   1:L PR[91] R[100]mm/sec CNT100;
   1:  PR[91,1] = PR[90,1] + 32.594;
   1:  PR[91,2] = PR[90,2] + 13.699;
   1:L PR[91] R[100]mm/sec CNT100;
   1:  PR[91,1] = PR[90,1] + 30.652;
   1:  PR[91,2] = PR[90,2] + 14.958;
   1:L PR[91] R[100]mm/sec CNT100;
   1:  PR[91,1] = PR[90,1] + 29.155;
   1:  PR[91,2] = PR[90,2] + 15.871;
   1:L PR[91] R[100]mm/sec CNT100;
   1:  PR[91,1] = PR[90,1] + 26.400;
   1:  PR[91,2] = PR[90,2] + 16.913;
   1:L PR[91] R[100]mm/sec CNT100;
   1:  PR[91,1] = PR[90,1] + 25.342;
   1:  PR[91,2] = PR[90,2] + 17.273;
   1:L PR[91] R[100]mm/sec CNT100;
   1:  PR[91,1] = PR[90,1] + 21.693;
   1:  PR[91,2] = PR[90,2] + 17.818;
   1:L PR[91] R[100]mm/sec CNT100;
   1:  PR[91,1] = PR[90,1] + 21.351;
   1:  PR[91,2] = PR[90,2] + 17.856;
   1:L PR[91] R[100]mm/sec CNT100;
   1:  PR[91,1] = PR[90,1] + 18.415;
   1:  PR[91,2] = PR[90,2] + 17.666;
   1:L PR[91] R[100]mm/sec CNT100;
   1:  PR[91,1] = PR[90,1] + 17.180;
   1:  PR[91,2] = PR[90,2] + 17.601;
   1:L PR[91] R[100]mm/sec CNT100;
   1:  PR[91,1] = PR[90,1] + 13.479;
   1:  PR[91,2] = PR[90,2] + 16.611;
   1:L PR[91] R[100]mm/sec CNT100;
   1:  PR[91,1] = PR[90,1] + 13.072;
   1:  PR[91,2] = PR[90,2] + 16.479;
   1:L PR[91] R[100]mm/sec CNT100;
   1:  PR[91,1] = PR[90,1] + 10.503;
   1:  PR[91,2] = PR[90,2] + 15.153;
   1:L PR[91] R[100]mm/sec CNT100;
   1:  PR[91,1] = PR[90,1] + 9.678;
   1:  PR[91,2] = PR[90,2] + 14.763;
   1:L PR[91] R[100]mm/sec CNT100;
   1:  PR[91,1] = PR[90,1] + 8.783;
   1:  PR[91,2] = PR[90,2] + 14.163;
   1:L PR[91] R[100]mm/sec CNT100;
   1:  PR[91,1] = PR[90,1] + 7.210;
   1:  PR[91,2] = PR[90,2] + 12.860;
   1:L PR[91] R[100]mm/sec CNT100;
   1:  PR[91,1] = PR[90,1] + 6.133;
   1:  PR[91,2] = PR[90,2] + 11.895;
   1:L PR[91] R[100]mm/sec CNT100;
   1:  PR[91,1] = PR[90,1] + 4.893;
   1:  PR[91,2] = PR[90,2] + 10.402;
   1:L PR[91] R[100]mm/sec CNT100;
   1:  PR[91,1] = PR[90,1] + 4.050;
   1:  PR[91,2] = PR[90,2] + 9.302;
   1:L PR[91] R[100]mm/sec CNT100;
   1:  PR[91,1] = PR[90,1] + 3.471;
   1:  PR[91,2] = PR[90,2] + 8.699;
   1:L PR[91] R[100]mm/sec CNT100;
   1:  PR[91,1] = PR[90,1] + 2.632;
   1:  PR[91,2] = PR[90,2] + 8.134;
   1:L PR[91] R[100]mm/sec CNT100;
   1:  PR[91,1] = PR[90,1] + 1.785;
   1:  PR[91,2] = PR[90,2] + 7.929;
   1:L PR[91] R[100]mm/sec CNT100;
   1:  PR[91,1] = PR[90,1] + 1.392;
   1:  PR[91,2] = PR[90,2] + 7.757;
   1:L PR[91] R[100]mm/sec CNT100;
   1:  PR[91] = PR[90];
   1:  PR[91,1] = PR[90,1] + -1.445;
   1:  PR[91,2] = PR[90,2] + 8.302;
   1:  PR[91,3] = PR[90,3] + 22.295;
   1:L PR[91] R[100]mm/sec CNT100;
   1:  PR[91,1] = PR[90,1] + -2.877;
   1:  PR[91,2] = PR[90,2] + 8.645;
   1:L PR[91] R[100]mm/sec CNT100;
   1:  PR[91,1] = PR[90,1] + -3.773;
   1:  PR[91,2] = PR[90,2] + 9.251;
   1:L PR[91] R[100]mm/sec CNT100;
   1:  PR[91,1] = PR[90,1] + -4.266;
   1:  PR[91,2] = PR[90,2] + 9.782;
   1:L PR[91] R[100]mm/sec CNT100;
   1:  PR[91,1] = PR[90,1] + -6.077;
   1:  PR[91,2] = PR[90,2] + 11.940;
   1:L PR[91] R[100]mm/sec CNT100;
   1:  PR[91,1] = PR[90,1] + -8.345;
   1:  PR[91,2] = PR[90,2] + 13.932;
   1:L PR[91] R[100]mm/sec CNT100;
   1:  PR[91,1] = PR[90,1] + -10.027;
   1:  PR[91,2] = PR[90,2] + 15.061;
   1:L PR[91] R[100]mm/sec CNT100;
   1:  PR[91,1] = PR[90,1] + -11.357;
   1:  PR[91,2] = PR[90,2] + 15.744;
   1:L PR[91] R[100]mm/sec CNT100;
   1:  PR[91,1] = PR[90,1] + -12.975;
   1:  PR[91,2] = PR[90,2] + 16.525;
   1:L PR[91] R[100]mm/sec CNT100;
   1:  PR[91,1] = PR[90,1] + -14.146;
   1:  PR[91,2] = PR[90,2] + 16.905;
   1:L PR[91] R[100]mm/sec CNT100;
   1:  PR[91,1] = PR[90,1] + -16.672;
   1:  PR[91,2] = PR[90,2] + 17.580;
   1:L PR[91] R[100]mm/sec CNT100;
   1:  PR[91,1] = PR[90,1] + -17.455;
   1:  PR[91,2] = PR[90,2] + 17.722;
   1:L PR[91] R[100]mm/sec CNT100;
   1:  PR[91,1] = PR[90,1] + -21.155;
   1:  PR[91,2] = PR[90,2] + 17.918;
   1:L PR[91] R[100]mm/sec CNT100;
   1:  PR[91,1] = PR[90,1] + -21.482;
   1:  PR[91,2] = PR[90,2] + 17.931;
   1:L PR[91] R[100]mm/sec CNT100;
   1:  PR[91,1] = PR[90,1] + -21.616;
   1:  PR[91,2] = PR[90,2] + 17.919;
   1:L PR[91] R[100]mm/sec CNT100;
   1:  PR[91,1] = PR[90,1] + -25.669;
   1:  PR[91,2] = PR[90,2] + 17.290;
   1:L PR[91] R[100]mm/sec CNT100;
   1:  PR[91,1] = PR[90,1] + -29.492;
   1:  PR[91,2] = PR[90,2] + 15.850;
   1:L PR[91] R[100]mm/sec CNT100;
   1:  PR[91,1] = PR[90,1] + -30.051;
   1:  PR[91,2] = PR[90,2] + 15.509;
   1:L PR[91] R[100]mm/sec CNT100;
   1:  PR[91,1] = PR[90,1] + -32.898;
   1:  PR[91,2] = PR[90,2] + 13.662;
   1:L PR[91] R[100]mm/sec CNT100;
   1:  PR[91,1] = PR[90,1] + -33.763;
   1:  PR[91,2] = PR[90,2] + 12.821;
   1:L PR[91] R[100]mm/sec CNT100;
   1:  PR[91,1] = PR[90,1] + -35.755;
   1:  PR[91,2] = PR[90,2] + 10.797;
   1:L PR[91] R[100]mm/sec CNT100;
   1:  PR[91,1] = PR[90,1] + -36.625;
   1:  PR[91,2] = PR[90,2] + 9.444;
   1:L PR[91] R[100]mm/sec CNT100;
   1:  PR[91,1] = PR[90,1] + -37.914;
   1:  PR[91,2] = PR[90,2] + 7.364;
   1:L PR[91] R[100]mm/sec CNT100;
   1:  PR[91,1] = PR[90,1] + -39.261;
   1:  PR[91,2] = PR[90,2] + 3.606;
   1:L PR[91] R[100]mm/sec CNT100;
   1:  PR[91,1] = PR[90,1] + -39.495;
   1:  PR[91,2] = PR[90,2] + 1.583;
   1:L PR[91] R[100]mm/sec CNT100;
   1:  PR[91,1] = PR[90,1] + -39.753;
   1:  PR[91,2] = PR[90,2] + -0.438;
   1:L PR[91] R[100]mm/sec CNT100;
   1:  PR[91,1] = PR[90,1] + -39.620;
   1:  PR[91,2] = PR[90,2] + -1.583;
   1:L PR[91] R[100]mm/sec CNT100;
   1:  PR[91,1] = PR[90,1] + -39.489;
   1:  PR[91,2] = PR[90,2] + -2.382;
   1:L PR[91] R[100]mm/sec CNT100;
   1:  PR[91,1] = PR[90,1] + -39.258;
   1:  PR[91,2] = PR[90,2] + -4.463;
   1:L PR[91] R[100]mm/sec CNT100;
   1:  PR[91,1] = PR[90,1] + -38.549;
   1:  PR[91,2] = PR[90,2] + -6.462;
   1:L PR[91] R[100]mm/sec CNT100;
   1:  PR[91,1] = PR[90,1] + -37.916;
   1:  PR[91,2] = PR[90,2] + -8.208;
   1:L PR[91] R[100]mm/sec CNT100;
   1:  PR[91,1] = PR[90,1] + -36.624;
   1:  PR[91,2] = PR[90,2] + -10.292;
   1:L PR[91] R[100]mm/sec CNT100;
   1:  PR[91,1] = PR[90,1] + -35.754;
   1:  PR[91,2] = PR[90,2] + -11.645;
   1:L PR[91] R[100]mm/sec CNT100;
   1:  PR[91,1] = PR[90,1] + -33.761;
   1:  PR[91,2] = PR[90,2] + -13.670;
   1:L PR[91] R[100]mm/sec CNT100;
   1:  PR[91,1] = PR[90,1] + -32.896;
   1:  PR[91,2] = PR[90,2] + -14.510;
   1:L PR[91] R[100]mm/sec CNT100;
   1:  PR[91,1] = PR[90,1] + -30.048;
   1:  PR[91,2] = PR[90,2] + -16.357;
   1:L PR[91] R[100]mm/sec CNT100;
   1:  PR[91,1] = PR[90,1] + -29.490;
   1:  PR[91,2] = PR[90,2] + -16.698;
   1:L PR[91] R[100]mm/sec CNT100;
   1:  PR[91,1] = PR[90,1] + -25.665;
   1:  PR[91,2] = PR[90,2] + -18.138;
   1:L PR[91] R[100]mm/sec CNT100;
   1:  PR[91,1] = PR[90,1] + -21.611;
   1:  PR[91,2] = PR[90,2] + -18.766;
   1:L PR[91] R[100]mm/sec CNT100;
   1:  PR[91,1] = PR[90,1] + -21.494;
   1:  PR[91,2] = PR[90,2] + -18.777;
   1:L PR[91] R[100]mm/sec CNT100;
   1:  PR[91,1] = PR[90,1] + -18.062;
   1:  PR[91,2] = PR[90,2] + -18.588;
   1:L PR[91] R[100]mm/sec CNT100;
   1:  PR[91,1] = PR[90,1] + -17.432;
   1:  PR[91,2] = PR[90,2] + -18.565;
   1:L PR[91] R[100]mm/sec CNT100;
   1:  PR[91,1] = PR[90,1] + -16.667;
   1:  PR[91,2] = PR[90,2] + -18.427;
   1:L PR[91] R[100]mm/sec CNT100;
   1:  PR[91,1] = PR[90,1] + -14.143;
   1:  PR[91,2] = PR[90,2] + -17.751;
   1:L PR[91] R[100]mm/sec CNT100;
   1:  PR[91,1] = PR[90,1] + -13.004;
   1:  PR[91,2] = PR[90,2] + -17.381;
   1:L PR[91] R[100]mm/sec CNT100;
   1:  PR[91,1] = PR[90,1] + -11.460;
   1:  PR[91,2] = PR[90,2] + -16.582;
   1:L PR[91] R[100]mm/sec CNT100;
   1:  PR[91,1] = PR[90,1] + -9.994;
   1:  PR[91,2] = PR[90,2] + -15.886;
   1:L PR[91] R[100]mm/sec CNT100;
   1:  PR[91,1] = PR[90,1] + -8.315;
   1:  PR[91,2] = PR[90,2] + -14.758;
   1:L PR[91] R[100]mm/sec CNT100;
   1:  PR[91,1] = PR[90,1] + -7.791;
   1:  PR[91,2] = PR[90,2] + -14.325;
   1:L PR[91] R[100]mm/sec CNT100;
   1:  PR[91,1] = PR[90,1] + -6.085;
   1:  PR[91,2] = PR[90,2] + -12.797;
   1:L PR[91] R[100]mm/sec CNT100;
   1:  PR[91,1] = PR[90,1] + -4.272;
   1:  PR[91,2] = PR[90,2] + -10.633;
   1:L PR[91] R[100]mm/sec CNT100;
   1:  PR[91,1] = PR[90,1] + -3.791;
   1:  PR[91,2] = PR[90,2] + -10.110;
   1:L PR[91] R[100]mm/sec CNT100;
   1:  PR[91,1] = PR[90,1] + -2.878;
   1:  PR[91,2] = PR[90,2] + -9.493;
   1:L PR[91] R[100]mm/sec CNT100;
   1:  PR[91,1] = PR[90,1] + -1.445;
   1:  PR[91,2] = PR[90,2] + -9.149;
   1:L PR[91] R[100]mm/sec CNT100;
   1:  PR[91,1] = PR[90,1] + 0.974;
   1:L PR[91] R[100]mm/sec CNT100;
   1:  PR[91,1] = PR[90,1] + 2.406;
   1:  PR[91,2] = PR[90,2] + -9.492;
   1:L PR[91] R[100]mm/sec CNT100;
   1:  PR[91,1] = PR[90,1] + 3.303;
   1:  PR[91,2] = PR[90,2] + -10.098;
   1:L PR[91] R[100]mm/sec CNT100;
   1:  PR[91,1] = PR[90,1] + 3.795;
   1:  PR[91,2] = PR[90,2] + -10.630;
   1:L PR[91] R[100]mm/sec CNT100;
   1:  PR[91,1] = PR[90,1] + 5.623;
   1:  PR[91,2] = PR[90,2] + -12.812;
   1:L PR[91] R[100]mm/sec CNT100;
   1:  PR[91,1] = PR[90,1] + 7.885;
   1:  PR[91,2] = PR[90,2] + -14.797;
   1:L PR[91] R[100]mm/sec CNT100;
   1:  PR[91,1] = PR[90,1] + 9.546;
   1:  PR[91,2] = PR[90,2] + -15.911;
   1:L PR[91] R[100]mm/sec CNT100;
   1:  PR[91,1] = PR[90,1] + 10.876;
   1:  PR[91,2] = PR[90,2] + -16.592;
   1:L PR[91] R[100]mm/sec CNT100;
   1:  PR[91,1] = PR[90,1] + 12.490;
   1:  PR[91,2] = PR[90,2] + -17.369;
   1:L PR[91] R[100]mm/sec CNT100;
   1:  PR[91,1] = PR[90,1] + 13.666;
   1:  PR[91,2] = PR[90,2] + -17.751;
   1:L PR[91] R[100]mm/sec CNT100;
   1:  PR[91,1] = PR[90,1] + 16.194;
   1:  PR[91,2] = PR[90,2] + -18.427;
   1:L PR[91] R[100]mm/sec CNT100;
   1:  PR[91,1] = PR[90,1] + 16.977;
   1:  PR[91,2] = PR[90,2] + -18.570;
   1:L PR[91] R[100]mm/sec CNT100;
   1:  PR[91,1] = PR[90,1] + 21.019;
   1:  PR[91,2] = PR[90,2] + -18.777;
   1:L PR[91] R[100]mm/sec CNT100;
   1:  PR[91,1] = PR[90,1] + 21.138;
   1:  PR[91,2] = PR[90,2] + -18.767;
   1:L PR[91] R[100]mm/sec CNT100;
   1:  PR[91,1] = PR[90,1] + 25.192;
   1:  PR[91,2] = PR[90,2] + -18.135;
   1:L PR[91] R[100]mm/sec CNT100;
   1:  PR[91,1] = PR[90,1] + 29.016;
   1:  PR[91,2] = PR[90,2] + -16.696;
   1:L PR[91] R[100]mm/sec CNT100;
   1:  PR[91,1] = PR[90,1] + 29.575;
   1:  PR[91,2] = PR[90,2] + -16.355;
   1:L PR[91] R[100]mm/sec CNT100;
   1:  PR[91,1] = PR[90,1] + 32.419;
   1:  PR[91,2] = PR[90,2] + -14.511;
   1:L PR[91] R[100]mm/sec CNT100;
   1:  PR[91,1] = PR[90,1] + 33.282;
   1:  PR[91,2] = PR[90,2] + -13.671;
   1:L PR[91] R[100]mm/sec CNT100;
   1:  PR[91,1] = PR[90,1] + 35.275;
   1:  PR[91,2] = PR[90,2] + -11.638;
   1:L PR[91] R[100]mm/sec CNT100;
   1:  PR[91,1] = PR[90,1] + 36.146;
   1:  PR[91,2] = PR[90,2] + -10.284;
   1:L PR[91] R[100]mm/sec CNT100;
   1:  PR[91,1] = PR[90,1] + 37.435;
   1:  PR[91,2] = PR[90,2] + -8.207;
   1:L PR[91] R[100]mm/sec CNT100;
   1:  PR[91,1] = PR[90,1] + 38.781;
   1:  PR[91,2] = PR[90,2] + -4.466;
   1:L PR[91] R[100]mm/sec CNT100;
   1:  PR[91,1] = PR[90,1] + 39.015;
   1:  PR[91,2] = PR[90,2] + -2.439;
   1:L PR[91] R[100]mm/sec CNT100;
   1:  PR[91,1] = PR[90,1] + 39.273;
   1:  PR[91,2] = PR[90,2] + -0.410;
   1:L PR[91] R[100]mm/sec CNT100;
   1:  PR[91,1] = PR[90,1] + 39.140;
   1:  PR[91,2] = PR[90,2] + 0.741;
   1:L PR[91] R[100]mm/sec CNT100;
   1:  PR[91,1] = PR[90,1] + 39.009;
   1:  PR[91,2] = PR[90,2] + 1.541;
   1:L PR[91] R[100]mm/sec CNT100;
   1:  PR[91,1] = PR[90,1] + 38.779;
   1:  PR[91,2] = PR[90,2] + 3.625;
   1:L PR[91] R[100]mm/sec CNT100;
   1:  PR[91,1] = PR[90,1] + 37.435;
   1:  PR[91,2] = PR[90,2] + 7.361;
   1:L PR[91] R[100]mm/sec CNT100;
   1:  PR[91,1] = PR[90,1] + 36.146;
   1:  PR[91,2] = PR[90,2] + 9.437;
   1:L PR[91] R[100]mm/sec CNT100;
   1:  PR[91,1] = PR[90,1] + 35.274;
   1:  PR[91,2] = PR[90,2] + 10.792;
   1:L PR[91] R[100]mm/sec CNT100;
   1:  PR[91,1] = PR[90,1] + 33.281;
   1:  PR[91,2] = PR[90,2] + 12.823;
   1:L PR[91] R[100]mm/sec CNT100;
   1:  PR[91,1] = PR[90,1] + 32.418;
   1:  PR[91,2] = PR[90,2] + 13.665;
   1:L PR[91] R[100]mm/sec CNT100;
   1:  PR[91,1] = PR[90,1] + 29.574;
   1:  PR[91,2] = PR[90,2] + 15.508;
   1:L PR[91] R[100]mm/sec CNT100;
   1:  PR[91,1] = PR[90,1] + 29.015;
   1:  PR[91,2] = PR[90,2] + 15.849;
   1:L PR[91] R[100]mm/sec CNT100;
   1:  PR[91,1] = PR[90,1] + 25.191;
   1:  PR[91,2] = PR[90,2] + 17.288;
   1:L PR[91] R[100]mm/sec CNT100;
   1:  PR[91,1] = PR[90,1] + 21.137;
   1:  PR[91,2] = PR[90,2] + 17.919;
   1:L PR[91] R[100]mm/sec CNT100;
   1:  PR[91,1] = PR[90,1] + 21.021;
   1:  PR[91,2] = PR[90,2] + 17.930;
   1:L PR[91] R[100]mm/sec CNT100;
   1:  PR[91,1] = PR[90,1] + 17.586;
   1:  PR[91,2] = PR[90,2] + 17.742;
   1:L PR[91] R[100]mm/sec CNT100;
   1:  PR[91,1] = PR[90,1] + 16.959;
   1:  PR[91,2] = PR[90,2] + 17.719;
   1:L PR[91] R[100]mm/sec CNT100;
   1:  PR[91,1] = PR[90,1] + 16.193;
   1:  PR[91,2] = PR[90,2] + 17.580;
   1:L PR[91] R[100]mm/sec CNT100;
   1:  PR[91,1] = PR[90,1] + 13.666;
   1:  PR[91,2] = PR[90,2] + 16.903;
   1:L PR[91] R[100]mm/sec CNT100;
   1:  PR[91,1] = PR[90,1] + 12.521;
   1:  PR[91,2] = PR[90,2] + 16.532;
   1:L PR[91] R[100]mm/sec CNT100;
   1:  PR[91,1] = PR[90,1] + 10.976;
   1:  PR[91,2] = PR[90,2] + 15.735;
   1:L PR[91] R[100]mm/sec CNT100;
   1:  PR[91,1] = PR[90,1] + 9.515;
   1:  PR[91,2] = PR[90,2] + 15.043;
   1:L PR[91] R[100]mm/sec CNT100;
   1:  PR[91,1] = PR[90,1] + 7.856;
   1:  PR[91,2] = PR[90,2] + 13.930;
   1:L PR[91] R[100]mm/sec CNT100;
   1:  PR[91,1] = PR[90,1] + 7.329;
   1:  PR[91,2] = PR[90,2] + 13.494;
   1:L PR[91] R[100]mm/sec CNT100;
   1:  PR[91,1] = PR[90,1] + 5.632;
   1:  PR[91,2] = PR[90,2] + 11.974;
   1:L PR[91] R[100]mm/sec CNT100;
   1:  PR[91,1] = PR[90,1] + 3.802;
   1:  PR[91,2] = PR[90,2] + 9.786;
   1:L PR[91] R[100]mm/sec CNT100;
   1:  PR[91,1] = PR[90,1] + 3.320;
   1:  PR[91,2] = PR[90,2] + 9.263;
   1:L PR[91] R[100]mm/sec CNT100;
   1:  PR[91,1] = PR[90,1] + 2.407;
   1:  PR[91,2] = PR[90,2] + 8.645;
   1:L PR[91] R[100]mm/sec CNT100;
   1:  PR[91,1] = PR[90,1] + 0.974;
   1:  PR[91,2] = PR[90,2] + 8.302;
   1:L PR[91] R[100]mm/sec CNT100;
   1:  PR[91] = PR[90];
   1:  PR[91,1] = PR[90,1] + -1.220;
   1:  PR[91,2] = PR[90,2] + 8.847;
   1:  PR[91,3] = PR[90,3] + 23.595;
   1:L PR[91] R[100]mm/sec CNT100;
   1:  PR[91,1] = PR[90,1] + -2.655;
   1:  PR[91,2] = PR[90,2] + 9.172;
   1:L PR[91] R[100]mm/sec CNT100;
   1:  PR[91,1] = PR[90,1] + -3.468;
   1:  PR[91,2] = PR[90,2] + 9.721;
   1:L PR[91] R[100]mm/sec CNT100;
   1:  PR[91,1] = PR[90,1] + -3.995;
   1:  PR[91,2] = PR[90,2] + 10.252;
   1:L PR[91] R[100]mm/sec CNT100;
   1:  PR[91,1] = PR[90,1] + -5.523;
   1:  PR[91,2] = PR[90,2] + 12.037;
   1:L PR[91] R[100]mm/sec CNT100;
   1:  PR[91,1] = PR[90,1] + -5.576;
   1:  PR[91,2] = PR[90,2] + 12.090;
   1:L PR[91] R[100]mm/sec CNT100;
   1:  PR[91,1] = PR[90,1] + -7.560;
   1:  PR[91,2] = PR[90,2] + 13.830;
   1:L PR[91] R[100]mm/sec CNT100;
   1:  PR[91,1] = PR[90,1] + -9.831;
   1:  PR[91,2] = PR[90,2] + 15.322;
   1:L PR[91] R[100]mm/sec CNT100;
   1:  PR[91,1] = PR[90,1] + -12.430;
   1:  PR[91,2] = PR[90,2] + 16.580;
   1:L PR[91] R[100]mm/sec CNT100;
   1:  PR[91,1] = PR[90,1] + -14.335;
   1:  PR[91,2] = PR[90,2] + 17.199;
   1:L PR[91] R[100]mm/sec CNT100;
   1:  PR[91,1] = PR[90,1] + -15.650;
   1:  PR[91,2] = PR[90,2] + 17.550;
   1:L PR[91] R[100]mm/sec CNT100;
   1:  PR[91,1] = PR[90,1] + -17.281;
   1:  PR[91,2] = PR[90,2] + 17.845;
   1:L PR[91] R[100]mm/sec CNT100;
   1:  PR[91,1] = PR[90,1] + -19.601;
   1:  PR[91,2] = PR[90,2] + 17.968;
   1:L PR[91] R[100]mm/sec CNT100;
   1:  PR[91,1] = PR[90,1] + -20.896;
   1:  PR[91,2] = PR[90,2] + 18.020;
   1:L PR[91] R[100]mm/sec CNT100;
   1:  PR[91,1] = PR[90,1] + -21.739;
   1:  PR[91,2] = PR[90,2] + 17.943;
   1:L PR[91] R[100]mm/sec CNT100;
   1:  PR[91,1] = PR[90,1] + -24.981;
   1:  PR[91,2] = PR[90,2] + 17.433;
   1:L PR[91] R[100]mm/sec CNT100;
   1:  PR[91,1] = PR[90,1] + -25.369;
   1:  PR[91,2] = PR[90,2] + 17.344;
   1:L PR[91] R[100]mm/sec CNT100;
   1:  PR[91,1] = PR[90,1] + -29.281;
   1:  PR[91,2] = PR[90,2] + 15.858;
   1:L PR[91] R[100]mm/sec CNT100;
   1:  PR[91,1] = PR[90,1] + -32.702;
   1:  PR[91,2] = PR[90,2] + 13.640;
   1:L PR[91] R[100]mm/sec CNT100;
   1:  PR[91,1] = PR[90,1] + -35.550;
   1:  PR[91,2] = PR[90,2] + 10.758;
   1:L PR[91] R[100]mm/sec CNT100;
   1:  PR[91,1] = PR[90,1] + -35.885;
   1:  PR[91,2] = PR[90,2] + 10.237;
   1:L PR[91] R[100]mm/sec CNT100;
   1:  PR[91,1] = PR[90,1] + -37.684;
   1:  PR[91,2] = PR[90,2] + 7.334;
   1:L PR[91] R[100]mm/sec CNT100;
   1:  PR[91,1] = PR[90,1] + -39.018;
   1:  PR[91,2] = PR[90,2] + 3.596;
   1:L PR[91] R[100]mm/sec CNT100;
   1:  PR[91,1] = PR[90,1] + -39.146;
   1:  PR[91,2] = PR[90,2] + 2.487;
   1:L PR[91] R[100]mm/sec CNT100;
   1:  PR[91,1] = PR[90,1] + -39.518;
   1:  PR[91,2] = PR[90,2] + -0.432;
   1:L PR[91] R[100]mm/sec CNT100;
   1:  PR[91,1] = PR[90,1] + -39.342;
   1:  PR[91,2] = PR[90,2] + -1.502;
   1:L PR[91] R[100]mm/sec CNT100;
   1:  PR[91,1] = PR[90,1] + -39.015;
   1:  PR[91,2] = PR[90,2] + -4.451;
   1:L PR[91] R[100]mm/sec CNT100;
   1:  PR[91,1] = PR[90,1] + -38.002;
   1:  PR[91,2] = PR[90,2] + -7.308;
   1:L PR[91] R[100]mm/sec CNT100;
   1:  PR[91,1] = PR[90,1] + -37.687;
   1:  PR[91,2] = PR[90,2] + -8.176;
   1:L PR[91] R[100]mm/sec CNT100;
   1:  PR[91,1] = PR[90,1] + -35.884;
   1:  PR[91,2] = PR[90,2] + -11.086;
   1:L PR[91] R[100]mm/sec CNT100;
   1:  PR[91,1] = PR[90,1] + -35.549;
   1:  PR[91,2] = PR[90,2] + -11.607;
   1:L PR[91] R[100]mm/sec CNT100;
   1:  PR[91,1] = PR[90,1] + -32.701;
   1:  PR[91,2] = PR[90,2] + -14.487;
   1:L PR[91] R[100]mm/sec CNT100;
   1:  PR[91,1] = PR[90,1] + -29.241;
   1:  PR[91,2] = PR[90,2] + -16.720;
   1:L PR[91] R[100]mm/sec CNT100;
   1:  PR[91,1] = PR[90,1] + -25.365;
   1:  PR[91,2] = PR[90,2] + -18.193;
   1:L PR[91] R[100]mm/sec CNT100;
   1:  PR[91,1] = PR[90,1] + -24.977;
   1:  PR[91,2] = PR[90,2] + -18.281;
   1:L PR[91] R[100]mm/sec CNT100;
   1:  PR[91,1] = PR[90,1] + -21.735;
   1:  PR[91,2] = PR[90,2] + -18.791;
   1:L PR[91] R[100]mm/sec CNT100;
   1:  PR[91,1] = PR[90,1] + -20.910;
   1:  PR[91,2] = PR[90,2] + -18.866;
   1:L PR[91] R[100]mm/sec CNT100;
   1:  PR[91,1] = PR[90,1] + -18.532;
   1:  PR[91,2] = PR[90,2] + -18.735;
   1:L PR[91] R[100]mm/sec CNT100;
   1:  PR[91,1] = PR[90,1] + -17.259;
   1:  PR[91,2] = PR[90,2] + -18.689;
   1:L PR[91] R[100]mm/sec CNT100;
   1:  PR[91,1] = PR[90,1] + -15.647;
   1:  PR[91,2] = PR[90,2] + -18.397;
   1:L PR[91] R[100]mm/sec CNT100;
   1:  PR[91,1] = PR[90,1] + -14.334;
   1:  PR[91,2] = PR[90,2] + -18.045;
   1:L PR[91] R[100]mm/sec CNT100;
   1:  PR[91,1] = PR[90,1] + -12.459;
   1:  PR[91,2] = PR[90,2] + -17.437;
   1:L PR[91] R[100]mm/sec CNT100;
   1:  PR[91,1] = PR[90,1] + -11.938;
   1:  PR[91,2] = PR[90,2] + -17.167;
   1:L PR[91] R[100]mm/sec CNT100;
   1:  PR[91,1] = PR[90,1] + -9.823;
   1:  PR[91,2] = PR[90,2] + -16.164;
   1:L PR[91] R[100]mm/sec CNT100;
   1:  PR[91,1] = PR[90,1] + -7.560;
   1:  PR[91,2] = PR[90,2] + -14.677;
   1:L PR[91] R[100]mm/sec CNT100;
   1:  PR[91,1] = PR[90,1] + -5.576;
   1:  PR[91,2] = PR[90,2] + -12.937;
   1:L PR[91] R[100]mm/sec CNT100;
   1:  PR[91,1] = PR[90,1] + -5.529;
   1:  PR[91,2] = PR[90,2] + -12.890;
   1:L PR[91] R[100]mm/sec CNT100;
   1:  PR[91,1] = PR[90,1] + -3.988;
   1:  PR[91,2] = PR[90,2] + -11.066;
   1:L PR[91] R[100]mm/sec CNT100;
   1:  PR[91,1] = PR[90,1] + -3.858;
   1:  PR[91,2] = PR[90,2] + -10.838;
   1:L PR[91] R[100]mm/sec CNT100;
   1:  PR[91,1] = PR[90,1] + -3.712;
   1:  PR[91,2] = PR[90,2] + -10.739;
   1:L PR[91] R[100]mm/sec CNT100;
   1:  PR[91,1] = PR[90,1] + -3.405;
   1:  PR[91,2] = PR[90,2] + -10.375;
   1:L PR[91] R[100]mm/sec CNT100;
   1:  PR[91,1] = PR[90,1] + -3.166;
   1:  PR[91,2] = PR[90,2] + -10.365;
   1:L PR[91] R[100]mm/sec CNT100;
   1:  PR[91,1] = PR[90,1] + -2.670;
   1:  PR[91,2] = PR[90,2] + -10.026;
   1:L PR[91] R[100]mm/sec CNT100;
   1:  PR[91,1] = PR[90,1] + -1.252;
   1:  PR[91,2] = PR[90,2] + -9.694;
   1:L PR[91] R[100]mm/sec CNT100;
   1:  PR[91,1] = PR[90,1] + 0.750;
   1:L PR[91] R[100]mm/sec CNT100;
   1:  PR[91,1] = PR[90,1] + 2.184;
   1:  PR[91,2] = PR[90,2] + -10.020;
   1:L PR[91] R[100]mm/sec CNT100;
   1:  PR[91,1] = PR[90,1] + 2.955;
   1:  PR[91,2] = PR[90,2] + -10.540;
   1:L PR[91] R[100]mm/sec CNT100;
   1:  PR[91,1] = PR[90,1] + 3.346;
   1:  PR[91,2] = PR[90,2] + -10.903;
   1:L PR[91] R[100]mm/sec CNT100;
   1:  PR[91,1] = PR[90,1] + 4.770;
   1:  PR[91,2] = PR[90,2] + -12.571;
   1:L PR[91] R[100]mm/sec CNT100;
   1:  PR[91,1] = PR[90,1] + 5.055;
   1:  PR[91,2] = PR[90,2] + -12.893;
   1:L PR[91] R[100]mm/sec CNT100;
   1:  PR[91,1] = PR[90,1] + 5.122;
   1:  PR[91,2] = PR[90,2] + -12.960;
   1:L PR[91] R[100]mm/sec CNT100;
   1:  PR[91,1] = PR[90,1] + 7.100;
   1:  PR[91,2] = PR[90,2] + -14.695;
   1:L PR[91] R[100]mm/sec CNT100;
   1:  PR[91,1] = PR[90,1] + 9.349;
   1:  PR[91,2] = PR[90,2] + -16.170;
   1:L PR[91] R[100]mm/sec CNT100;
   1:  PR[91,1] = PR[90,1] + 11.940;
   1:  PR[91,2] = PR[90,2] + -17.422;
   1:L PR[91] R[100]mm/sec CNT100;
   1:  PR[91,1] = PR[90,1] + 13.853;
   1:  PR[91,2] = PR[90,2] + -18.044;
   1:L PR[91] R[100]mm/sec CNT100;
   1:  PR[91,1] = PR[90,1] + 15.168;
   1:  PR[91,2] = PR[90,2] + -18.395;
   1:L PR[91] R[100]mm/sec CNT100;
   1:  PR[91,1] = PR[90,1] + 16.802;
   1:  PR[91,2] = PR[90,2] + -18.693;
   1:L PR[91] R[100]mm/sec CNT100;
   1:  PR[91,1] = PR[90,1] + 19.122;
   1:  PR[91,2] = PR[90,2] + -18.815;
   1:L PR[91] R[100]mm/sec CNT100;
   1:  PR[91,1] = PR[90,1] + 20.414;
   1:  PR[91,2] = PR[90,2] + -18.867;
   1:L PR[91] R[100]mm/sec CNT100;
   1:  PR[91,1] = PR[90,1] + 21.253;
   1:  PR[91,2] = PR[90,2] + -18.792;
   1:L PR[91] R[100]mm/sec CNT100;
   1:  PR[91,1] = PR[90,1] + 24.497;
   1:  PR[91,2] = PR[90,2] + -18.280;
   1:L PR[91] R[100]mm/sec CNT100;
   1:  PR[91,1] = PR[90,1] + 24.887;
   1:  PR[91,2] = PR[90,2] + -18.191;
   1:L PR[91] R[100]mm/sec CNT100;
   1:  PR[91,1] = PR[90,1] + 28.767;
   1:  PR[91,2] = PR[90,2] + -16.718;
   1:L PR[91] R[100]mm/sec CNT100;
   1:  PR[91,1] = PR[90,1] + 32.224;
   1:  PR[91,2] = PR[90,2] + -14.488;
   1:L PR[91] R[100]mm/sec CNT100;
   1:  PR[91,1] = PR[90,1] + 35.070;
   1:  PR[91,2] = PR[90,2] + -11.598;
   1:L PR[91] R[100]mm/sec CNT100;
   1:  PR[91,1] = PR[90,1] + 35.407;
   1:  PR[91,2] = PR[90,2] + -11.075;
   1:L PR[91] R[100]mm/sec CNT100;
   1:  PR[91,1] = PR[90,1] + 37.206;
   1:  PR[91,2] = PR[90,2] + -8.177;
   1:L PR[91] R[100]mm/sec CNT100;
   1:  PR[91,1] = PR[90,1] + 38.538;
   1:  PR[91,2] = PR[90,2] + -4.457;
   1:L PR[91] R[100]mm/sec CNT100;
   1:  PR[91,1] = PR[90,1] + 38.666;
   1:  PR[91,2] = PR[90,2] + -3.347;
   1:L PR[91] R[100]mm/sec CNT100;
   1:  PR[91,1] = PR[90,1] + 39.039;
   1:  PR[91,2] = PR[90,2] + -0.415;
   1:L PR[91] R[100]mm/sec CNT100;
   1:  PR[91,1] = PR[90,1] + 38.863;
   1:  PR[91,2] = PR[90,2] + 0.659;
   1:L PR[91] R[100]mm/sec CNT100;
   1:  PR[91,1] = PR[90,1] + 38.536;
   1:  PR[91,2] = PR[90,2] + 3.616;
   1:L PR[91] R[100]mm/sec CNT100;
   1:  PR[91,1] = PR[90,1] + 37.206;
   1:  PR[91,2] = PR[90,2] + 7.330;
   1:L PR[91] R[100]mm/sec CNT100;
   1:  PR[91,1] = PR[90,1] + 35.407;
   1:  PR[91,2] = PR[90,2] + 10.229;
   1:L PR[91] R[100]mm/sec CNT100;
   1:  PR[91,1] = PR[90,1] + 35.069;
   1:  PR[91,2] = PR[90,2] + 10.754;
   1:L PR[91] R[100]mm/sec CNT100;
   1:  PR[91,1] = PR[90,1] + 32.363;
   1:  PR[91,2] = PR[90,2] + 13.513;
   1:L PR[91] R[100]mm/sec CNT100;
   1:  PR[91,1] = PR[90,1] + 32.244;
   1:  PR[91,2] = PR[90,2] + 13.628;
   1:L PR[91] R[100]mm/sec CNT100;
   1:  PR[91,1] = PR[90,1] + 28.767;
   1:  PR[91,2] = PR[90,2] + 15.871;
   1:L PR[91] R[100]mm/sec CNT100;
   1:  PR[91,1] = PR[90,1] + 24.887;
   1:  PR[91,2] = PR[90,2] + 17.344;
   1:L PR[91] R[100]mm/sec CNT100;
   1:  PR[91,1] = PR[90,1] + 24.496;
   1:  PR[91,2] = PR[90,2] + 17.433;
   1:L PR[91] R[100]mm/sec CNT100;
   1:  PR[91,1] = PR[90,1] + 21.253;
   1:  PR[91,2] = PR[90,2] + 17.945;
   1:L PR[91] R[100]mm/sec CNT100;
   1:  PR[91,1] = PR[90,1] + 20.430;
   1:  PR[91,2] = PR[90,2] + 18.019;
   1:L PR[91] R[100]mm/sec CNT100;
   1:  PR[91,1] = PR[90,1] + 18.050;
   1:  PR[91,2] = PR[90,2] + 17.889;
   1:L PR[91] R[100]mm/sec CNT100;
   1:  PR[91,1] = PR[90,1] + 16.783;
   1:  PR[91,2] = PR[90,2] + 17.842;
   1:L PR[91] R[100]mm/sec CNT100;
   1:  PR[91,1] = PR[90,1] + 15.168;
   1:  PR[91,2] = PR[90,2] + 17.548;
   1:L PR[91] R[100]mm/sec CNT100;
   1:  PR[91,1] = PR[90,1] + 13.853;
   1:  PR[91,2] = PR[90,2] + 17.196;
   1:L PR[91] R[100]mm/sec CNT100;
   1:  PR[91,1] = PR[90,1] + 11.970;
   1:  PR[91,2] = PR[90,2] + 16.585;
   1:L PR[91] R[100]mm/sec CNT100;
   1:  PR[91,1] = PR[90,1] + 11.449;
   1:  PR[91,2] = PR[90,2] + 16.316;
   1:L PR[91] R[100]mm/sec CNT100;
   1:  PR[91,1] = PR[90,1] + 9.341;
   1:  PR[91,2] = PR[90,2] + 15.318;
   1:L PR[91] R[100]mm/sec CNT100;
   1:  PR[91,1] = PR[90,1] + 7.100;
   1:  PR[91,2] = PR[90,2] + 13.848;
   1:L PR[91] R[100]mm/sec CNT100;
   1:  PR[91,1] = PR[90,1] + 5.122;
   1:  PR[91,2] = PR[90,2] + 12.113;
   1:L PR[91] R[100]mm/sec CNT100;
   1:  PR[91,1] = PR[90,1] + 5.075;
   1:  PR[91,2] = PR[90,2] + 12.066;
   1:L PR[91] R[100]mm/sec CNT100;
   1:  PR[91,1] = PR[90,1] + 3.580;
   1:  PR[91,2] = PR[90,2] + 10.293;
   1:L PR[91] R[100]mm/sec CNT100;
   1:  PR[91,1] = PR[90,1] + 3.158;
   1:  PR[91,2] = PR[90,2] + 9.836;
   1:L PR[91] R[100]mm/sec CNT100;
   1:  PR[91,1] = PR[90,1] + 2.198;
   1:  PR[91,2] = PR[90,2] + 9.179;
   1:L PR[91] R[100]mm/sec CNT100;
   1:  PR[91,1] = PR[90,1] + 0.780;
   1:  PR[91,2] = PR[90,2] + 8.847;
   1:L PR[91] R[100]mm/sec CNT100;
   1:  PR[91] = PR[90];
   1:  PR[91,1] = PR[90,1] + -0.996;
   1:  PR[91,2] = PR[90,2] + 9.391;
   1:  PR[91,3] = PR[90,3] + 24.895;
   1:L PR[91] R[100]mm/sec CNT100;
   1:  PR[91,1] = PR[90,1] + -2.434;
   1:  PR[91,2] = PR[90,2] + 9.699;
   1:L PR[91] R[100]mm/sec CNT100;
   1:  PR[91,1] = PR[90,1] + -3.156;
   1:  PR[91,2] = PR[90,2] + 10.187;
   1:L PR[91] R[100]mm/sec CNT100;
   1:  PR[91,1] = PR[90,1] + -3.672;
   1:  PR[91,2] = PR[90,2] + 10.667;
   1:L PR[91] R[100]mm/sec CNT100;
   1:  PR[91,1] = PR[90,1] + -4.901;
   1:  PR[91,2] = PR[90,2] + 12.071;
   1:L PR[91] R[100]mm/sec CNT100;
   1:  PR[91,1] = PR[90,1] + -5.179;
   1:  PR[91,2] = PR[90,2] + 12.346;
   1:L PR[91] R[100]mm/sec CNT100;
   1:  PR[91,1] = PR[90,1] + -7.039;
   1:  PR[91,2] = PR[90,2] + 13.969;
   1:L PR[91] R[100]mm/sec CNT100;
   1:  PR[91,1] = PR[90,1] + -9.174;
   1:  PR[91,2] = PR[90,2] + 15.363;
   1:L PR[91] R[100]mm/sec CNT100;
   1:  PR[91,1] = PR[90,1] + -9.436;
   1:  PR[91,2] = PR[90,2] + 15.511;
   1:L PR[91] R[100]mm/sec CNT100;
   1:  PR[91,1] = PR[90,1] + -11.840;
   1:  PR[91,2] = PR[90,2] + 16.641;
   1:L PR[91] R[100]mm/sec CNT100;
   1:  PR[91,1] = PR[90,1] + -14.518;
   1:  PR[91,2] = PR[90,2] + 17.490;
   1:L PR[91] R[100]mm/sec CNT100;
   1:  PR[91,1] = PR[90,1] + -14.627;
   1:  PR[91,2] = PR[90,2] + 17.520;
   1:L PR[91] R[100]mm/sec CNT100;
   1:  PR[91,1] = PR[90,1] + -17.097;
   1:  PR[91,2] = PR[90,2] + 17.966;
   1:L PR[91] R[100]mm/sec CNT100;
   1:  PR[91,1] = PR[90,1] + -20.315;
   1:  PR[91,2] = PR[90,2] + 18.108;
   1:L PR[91] R[100]mm/sec CNT100;
   1:  PR[91,1] = PR[90,1] + -21.864;
   1:  PR[91,2] = PR[90,2] + 17.967;
   1:L PR[91] R[100]mm/sec CNT100;
   1:  PR[91,1] = PR[90,1] + -23.973;
   1:  PR[91,2] = PR[90,2] + 17.636;
   1:L PR[91] R[100]mm/sec CNT100;
   1:  PR[91,1] = PR[90,1] + -25.128;
   1:  PR[91,2] = PR[90,2] + 17.372;
   1:L PR[91] R[100]mm/sec CNT100;
   1:  PR[91,1] = PR[90,1] + -28.742;
   1:  PR[91,2] = PR[90,2] + 15.997;
   1:L PR[91] R[100]mm/sec CNT100;
   1:  PR[91,1] = PR[90,1] + -29.203;
   1:  PR[91,2] = PR[90,2] + 15.747;
   1:L PR[91] R[100]mm/sec CNT100;
   1:  PR[91,1] = PR[90,1] + -32.278;
   1:  PR[91,2] = PR[90,2] + 13.758;
   1:L PR[91] R[100]mm/sec CNT100;
   1:  PR[91,1] = PR[90,1] + -32.405;
   1:  PR[91,2] = PR[90,2] + 13.665;
   1:L PR[91] R[100]mm/sec CNT100;
   1:  PR[91,1] = PR[90,1] + -35.302;
   1:  PR[91,2] = PR[90,2] + 10.756;
   1:L PR[91] R[100]mm/sec CNT100;
   1:  PR[91,1] = PR[90,1] + -37.456;
   1:  PR[91,2] = PR[90,2] + 7.301;
   1:L PR[91] R[100]mm/sec CNT100;
   1:  PR[91,1] = PR[90,1] + -38.778;
   1:  PR[91,2] = PR[90,2] + 3.575;
   1:L PR[91] R[100]mm/sec CNT100;
   1:  PR[91,1] = PR[90,1] + -38.972;
   1:  PR[91,2] = PR[90,2] + 2.019;
   1:L PR[91] R[100]mm/sec CNT100;
   1:  PR[91,1] = PR[90,1] + -39.239;
   1:  PR[91,2] = PR[90,2] + -0.361;
   1:L PR[91] R[100]mm/sec CNT100;
   1:  PR[91,1] = PR[90,1] + -39.196;
   1:  PR[91,2] = PR[90,2] + -0.623;
   1:L PR[91] R[100]mm/sec CNT100;
   1:  PR[91,1] = PR[90,1] + -38.773;
   1:  PR[91,2] = PR[90,2] + -4.439;
   1:L PR[91] R[100]mm/sec CNT100;
   1:  PR[91,1] = PR[90,1] + -37.459;
   1:  PR[91,2] = PR[90,2] + -8.142;
   1:L PR[91] R[100]mm/sec CNT100;
   1:  PR[91,1] = PR[90,1] + -35.300;
   1:  PR[91,2] = PR[90,2] + -11.605;
   1:L PR[91] R[100]mm/sec CNT100;
   1:  PR[91,1] = PR[90,1] + -32.403;
   1:  PR[91,2] = PR[90,2] + -14.513;
   1:L PR[91] R[100]mm/sec CNT100;
   1:  PR[91,1] = PR[90,1] + -32.276;
   1:  PR[91,2] = PR[90,2] + -14.607;
   1:L PR[91] R[100]mm/sec CNT100;
   1:  PR[91,1] = PR[90,1] + -29.201;
   1:  PR[91,2] = PR[90,2] + -16.596;
   1:L PR[91] R[100]mm/sec CNT100;
   1:  PR[91,1] = PR[90,1] + -28.739;
   1:  PR[91,2] = PR[90,2] + -16.845;
   1:L PR[91] R[100]mm/sec CNT100;
   1:  PR[91,1] = PR[90,1] + -25.126;
   1:  PR[91,2] = PR[90,2] + -18.220;
   1:L PR[91] R[100]mm/sec CNT100;
   1:  PR[91,1] = PR[90,1] + -23.970;
   1:  PR[91,2] = PR[90,2] + -18.483;
   1:L PR[91] R[100]mm/sec CNT100;
   1:  PR[91,1] = PR[90,1] + -21.861;
   1:  PR[91,2] = PR[90,2] + -18.815;
   1:L PR[91] R[100]mm/sec CNT100;
   1:  PR[91,1] = PR[90,1] + -20.326;
   1:  PR[91,2] = PR[90,2] + -18.954;
   1:L PR[91] R[100]mm/sec CNT100;
   1:  PR[91,1] = PR[90,1] + -19.002;
   1:  PR[91,2] = PR[90,2] + -18.882;
   1:L PR[91] R[100]mm/sec CNT100;
   1:  PR[91,1] = PR[90,1] + -17.087;
   1:  PR[91,2] = PR[90,2] + -18.812;
   1:L PR[91] R[100]mm/sec CNT100;
   1:  PR[91,1] = PR[90,1] + -14.627;
   1:  PR[91,2] = PR[90,2] + -18.367;
   1:L PR[91] R[100]mm/sec CNT100;
   1:  PR[91,1] = PR[90,1] + -14.518;
   1:  PR[91,2] = PR[90,2] + -18.337;
   1:L PR[91] R[100]mm/sec CNT100;
   1:  PR[91,1] = PR[90,1] + -11.840;
   1:  PR[91,2] = PR[90,2] + -17.488;
   1:L PR[91] R[100]mm/sec CNT100;
   1:  PR[91,1] = PR[90,1] + -9.436;
   1:  PR[91,2] = PR[90,2] + -16.358;
   1:L PR[91] R[100]mm/sec CNT100;
   1:  PR[91,1] = PR[90,1] + -9.173;
   1:  PR[91,2] = PR[90,2] + -16.210;
   1:L PR[91] R[100]mm/sec CNT100;
   1:  PR[91,1] = PR[90,1] + -7.038;
   1:  PR[91,2] = PR[90,2] + -14.815;
   1:L PR[91] R[100]mm/sec CNT100;
   1:  PR[91,1] = PR[90,1] + -5.178;
   1:  PR[91,2] = PR[90,2] + -13.193;
   1:L PR[91] R[100]mm/sec CNT100;
   1:  PR[91,1] = PR[90,1] + -4.917;
   1:  PR[91,2] = PR[90,2] + -12.933;
   1:L PR[91] R[100]mm/sec CNT100;
   1:  PR[91,1] = PR[90,1] + -3.832;
   1:  PR[91,2] = PR[90,2] + -11.649;
   1:L PR[91] R[100]mm/sec CNT100;
   1:  PR[91,1] = PR[90,1] + -3.695;
   1:  PR[91,2] = PR[90,2] + -11.410;
   1:L PR[91] R[100]mm/sec CNT100;
   1:  PR[91,1] = PR[90,1] + -3.540;
   1:  PR[91,2] = PR[90,2] + -11.303;
   1:L PR[91] R[100]mm/sec CNT100;
   1:  PR[91,1] = PR[90,1] + -3.187;
   1:  PR[91,2] = PR[90,2] + -10.886;
   1:L PR[91] R[100]mm/sec CNT100;
   1:  PR[91,1] = PR[90,1] + -2.918;
   1:  PR[91,2] = PR[90,2] + -10.874;
   1:L PR[91] R[100]mm/sec CNT100;
   1:  PR[91,1] = PR[90,1] + -2.459;
   1:  PR[91,2] = PR[90,2] + -10.558;
   1:L PR[91] R[100]mm/sec CNT100;
   1:  PR[91,1] = PR[90,1] + -1.055;
   1:  PR[91,2] = PR[90,2] + -10.238;
   1:L PR[91] R[100]mm/sec CNT100;
   1:  PR[91,1] = PR[90,1] + 0.525;
   1:L PR[91] R[100]mm/sec CNT100;
   1:  PR[91,1] = PR[90,1] + 1.962;
   1:  PR[91,2] = PR[90,2] + -10.547;
   1:L PR[91] R[100]mm/sec CNT100;
   1:  PR[91,1] = PR[90,1] + 2.682;
   1:  PR[91,2] = PR[90,2] + -11.033;
   1:L PR[91] R[100]mm/sec CNT100;
   1:  PR[91,1] = PR[90,1] + 3.200;
   1:  PR[91,2] = PR[90,2] + -11.514;
   1:L PR[91] R[100]mm/sec CNT100;
   1:  PR[91,1] = PR[90,1] + 4.443;
   1:  PR[91,2] = PR[90,2] + -12.937;
   1:L PR[91] R[100]mm/sec CNT100;
   1:  PR[91,1] = PR[90,1] + 4.721;
   1:  PR[91,2] = PR[90,2] + -13.213;
   1:L PR[91] R[100]mm/sec CNT100;
   1:  PR[91,1] = PR[90,1] + 6.576;
   1:  PR[91,2] = PR[90,2] + -14.832;
   1:L PR[91] R[100]mm/sec CNT100;
   1:  PR[91,1] = PR[90,1] + 8.691;
   1:  PR[91,2] = PR[90,2] + -16.212;
   1:L PR[91] R[100]mm/sec CNT100;
   1:  PR[91,1] = PR[90,1] + 8.953;
   1:  PR[91,2] = PR[90,2] + -16.359;
   1:L PR[91] R[100]mm/sec CNT100;
   1:  PR[91,1] = PR[90,1] + 11.348;
   1:  PR[91,2] = PR[90,2] + -17.482;
   1:L PR[91] R[100]mm/sec CNT100;
   1:  PR[91,1] = PR[90,1] + 14.032;
   1:  PR[91,2] = PR[90,2] + -18.334;
   1:L PR[91] R[100]mm/sec CNT100;
   1:  PR[91,1] = PR[90,1] + 14.142;
   1:  PR[91,2] = PR[90,2] + -18.363;
   1:L PR[91] R[100]mm/sec CNT100;
   1:  PR[91,1] = PR[90,1] + 16.615;
   1:  PR[91,2] = PR[90,2] + -18.814;
   1:L PR[91] R[100]mm/sec CNT100;
   1:  PR[91,1] = PR[90,1] + 19.827;
   1:  PR[91,2] = PR[90,2] + -18.956;
   1:L PR[91] R[100]mm/sec CNT100;
   1:  PR[91,1] = PR[90,1] + 21.371;
   1:  PR[91,2] = PR[90,2] + -18.817;
   1:L PR[91] R[100]mm/sec CNT100;
   1:  PR[91,1] = PR[90,1] + 23.479;
   1:  PR[91,2] = PR[90,2] + -18.484;
   1:L PR[91] R[100]mm/sec CNT100;
   1:  PR[91,1] = PR[90,1] + 24.640;
   1:  PR[91,2] = PR[90,2] + -18.220;
   1:L PR[91] R[100]mm/sec CNT100;
   1:  PR[91,1] = PR[90,1] + 28.262;
   1:  PR[91,2] = PR[90,2] + -16.845;
   1:L PR[91] R[100]mm/sec CNT100;
   1:  PR[91,1] = PR[90,1] + 28.722;
   1:  PR[91,2] = PR[90,2] + -16.597;
   1:L PR[91] R[100]mm/sec CNT100;
   1:  PR[91,1] = PR[90,1] + 31.798;
   1:  PR[91,2] = PR[90,2] + -14.609;
   1:L PR[91] R[100]mm/sec CNT100;
   1:  PR[91,1] = PR[90,1] + 31.920;
   1:  PR[91,2] = PR[90,2] + -14.519;
   1:L PR[91] R[100]mm/sec CNT100;
   1:  PR[91,1] = PR[90,1] + 34.857;
   1:  PR[91,2] = PR[90,2] + -11.551;
   1:L PR[91] R[100]mm/sec CNT100;
   1:  PR[91,1] = PR[90,1] + 36.977;
   1:  PR[91,2] = PR[90,2] + -8.146;
   1:L PR[91] R[100]mm/sec CNT100;
   1:  PR[91,1] = PR[90,1] + 38.298;
   1:  PR[91,2] = PR[90,2] + -4.438;
   1:L PR[91] R[100]mm/sec CNT100;
   1:  PR[91,1] = PR[90,1] + 38.492;
   1:  PR[91,2] = PR[90,2] + -2.877;
   1:L PR[91] R[100]mm/sec CNT100;
   1:  PR[91,1] = PR[90,1] + 38.759;
   1:  PR[91,2] = PR[90,2] + -0.486;
   1:L PR[91] R[100]mm/sec CNT100;
   1:  PR[91,1] = PR[90,1] + 38.716;
   1:  PR[91,2] = PR[90,2] + -0.222;
   1:L PR[91] R[100]mm/sec CNT100;
   1:  PR[91,1] = PR[90,1] + 38.293;
   1:  PR[91,2] = PR[90,2] + 3.607;
   1:L PR[91] R[100]mm/sec CNT100;
   1:  PR[91,1] = PR[90,1] + 36.977;
   1:  PR[91,2] = PR[90,2] + 7.297;
   1:L PR[91] R[100]mm/sec CNT100;
   1:  PR[91,1] = PR[90,1] + 34.821;
   1:  PR[91,2] = PR[90,2] + 10.751;
   1:L PR[91] R[100]mm/sec CNT100;
   1:  PR[91,1] = PR[90,1] + 32.041;
   1:  PR[91,2] = PR[90,2] + 13.558;
   1:L PR[91] R[100]mm/sec CNT100;
   1:  PR[91,1] = PR[90,1] + 31.936;
   1:  PR[91,2] = PR[90,2] + 13.660;
   1:L PR[91] R[100]mm/sec CNT100;
   1:  PR[91,1] = PR[90,1] + 31.797;
   1:  PR[91,2] = PR[90,2] + 13.762;
   1:L PR[91] R[100]mm/sec CNT100;
   1:  PR[91,1] = PR[90,1] + 28.721;
   1:  PR[91,2] = PR[90,2] + 15.750;
   1:L PR[91] R[100]mm/sec CNT100;
   1:  PR[91,1] = PR[90,1] + 28.261;
   1:  PR[91,2] = PR[90,2] + 15.998;
   1:L PR[91] R[100]mm/sec CNT100;
   1:  PR[91,1] = PR[90,1] + 24.639;
   1:  PR[91,2] = PR[90,2] + 17.373;
   1:L PR[91] R[100]mm/sec CNT100;
   1:  PR[91,1] = PR[90,1] + 23.478;
   1:  PR[91,2] = PR[90,2] + 17.637;
   1:L PR[91] R[100]mm/sec CNT100;
   1:  PR[91,1] = PR[90,1] + 21.371;
   1:  PR[91,2] = PR[90,2] + 17.970;
   1:L PR[91] R[100]mm/sec CNT100;
   1:  PR[91,1] = PR[90,1] + 19.839;
   1:  PR[91,2] = PR[90,2] + 18.108;
   1:L PR[91] R[100]mm/sec CNT100;
   1:  PR[91,1] = PR[90,1] + 18.515;
   1:  PR[91,2] = PR[90,2] + 18.036;
   1:L PR[91] R[100]mm/sec CNT100;
   1:  PR[91,1] = PR[90,1] + 16.606;
   1:  PR[91,2] = PR[90,2] + 17.965;
   1:L PR[91] R[100]mm/sec CNT100;
   1:  PR[91,1] = PR[90,1] + 14.142;
   1:  PR[91,2] = PR[90,2] + 17.516;
   1:L PR[91] R[100]mm/sec CNT100;
   1:  PR[91,1] = PR[90,1] + 14.033;
   1:  PR[91,2] = PR[90,2] + 17.487;
   1:L PR[91] R[100]mm/sec CNT100;
   1:  PR[91,1] = PR[90,1] + 11.348;
   1:  PR[91,2] = PR[90,2] + 16.635;
   1:L PR[91] R[100]mm/sec CNT100;
   1:  PR[91,1] = PR[90,1] + 8.953;
   1:  PR[91,2] = PR[90,2] + 15.512;
   1:L PR[91] R[100]mm/sec CNT100;
   1:  PR[91,1] = PR[90,1] + 8.691;
   1:  PR[91,2] = PR[90,2] + 15.365;
   1:L PR[91] R[100]mm/sec CNT100;
   1:  PR[91,1] = PR[90,1] + 6.553;
   1:  PR[91,2] = PR[90,2] + 13.971;
   1:L PR[91] R[100]mm/sec CNT100;
   1:  PR[91,1] = PR[90,1] + 6.419;
   1:  PR[91,2] = PR[90,2] + 13.859;
   1:L PR[91] R[100]mm/sec CNT100;
   1:  PR[91,1] = PR[90,1] + 4.724;
   1:  PR[91,2] = PR[90,2] + 12.369;
   1:L PR[91] R[100]mm/sec CNT100;
   1:  PR[91,1] = PR[90,1] + 4.454;
   1:  PR[91,2] = PR[90,2] + 12.100;
   1:L PR[91] R[100]mm/sec CNT100;
   1:  PR[91,1] = PR[90,1] + 3.042;
   1:  PR[91,2] = PR[90,2] + 10.442;
   1:L PR[91] R[100]mm/sec CNT100;
   1:  PR[91,1] = PR[90,1] + 2.547;
   1:  PR[91,2] = PR[90,2] + 10.095;
   1:L PR[91] R[100]mm/sec CNT100;
   1:  PR[91,1] = PR[90,1] + 1.974;
   1:  PR[91,2] = PR[90,2] + 9.708;
   1:L PR[91] R[100]mm/sec CNT100;
   1:  PR[91,1] = PR[90,1] + 0.582;
   1:  PR[91,2] = PR[90,2] + 9.391;
   1:L PR[91] R[100]mm/sec CNT100;
   1:  PR[91] = PR[90];
   1:  PR[91,1] = PR[90,1] + -0.800;
   1:  PR[91,2] = PR[90,2] + 9.936;
   1:  PR[91,3] = PR[90,3] + 26.195;
   1:L PR[91] R[100]mm/sec CNT100;
   1:  PR[91,1] = PR[90,1] + -2.218;
   1:  PR[91,2] = PR[90,2] + 10.230;
   1:L PR[91] R[100]mm/sec CNT100;
   1:  PR[91,1] = PR[90,1] + -2.885;
   1:  PR[91,2] = PR[90,2] + 10.680;
   1:L PR[91] R[100]mm/sec CNT100;
   1:  PR[91,1] = PR[90,1] + -3.169;
   1:  PR[91,2] = PR[90,2] + 10.945;
   1:L PR[91] R[100]mm/sec CNT100;
   1:  PR[91,1] = PR[90,1] + -3.383;
   1:  PR[91,2] = PR[90,2] + 11.094;
   1:L PR[91] R[100]mm/sec CNT100;
   1:  PR[91,1] = PR[90,1] + -4.283;
   1:  PR[91,2] = PR[90,2] + 12.109;
   1:L PR[91] R[100]mm/sec CNT100;
   1:  PR[91,1] = PR[90,1] + -4.787;
   1:  PR[91,2] = PR[90,2] + 12.607;
   1:L PR[91] R[100]mm/sec CNT100;
   1:  PR[91,1] = PR[90,1] + -6.171;
   1:  PR[91,2] = PR[90,2] + 13.824;
   1:L PR[91] R[100]mm/sec CNT100;
   1:  PR[91,1] = PR[90,1] + -6.499;
   1:  PR[91,2] = PR[90,2] + 14.097;
   1:L PR[91] R[100]mm/sec CNT100;
   1:  PR[91,1] = PR[90,1] + -8.389;
   1:  PR[91,2] = PR[90,2] + 15.331;
   1:L PR[91] R[100]mm/sec CNT100;
   1:  PR[91,1] = PR[90,1] + -9.110;
   1:  PR[91,2] = PR[90,2] + 15.737;
   1:L PR[91] R[100]mm/sec CNT100;
   1:  PR[91,1] = PR[90,1] + -11.224;
   1:  PR[91,2] = PR[90,2] + 16.730;
   1:L PR[91] R[100]mm/sec CNT100;
   1:  PR[91,1] = PR[90,1] + -14.122;
   1:  PR[91,2] = PR[90,2] + 17.635;
   1:L PR[91] R[100]mm/sec CNT100;
   1:  PR[91,1] = PR[90,1] + -16.789;
   1:  PR[91,2] = PR[90,2] + 18.082;
   1:L PR[91] R[100]mm/sec CNT100;
   1:  PR[91,1] = PR[90,1] + -19.724;
   1:  PR[91,2] = PR[90,2] + 18.198;
   1:L PR[91] R[100]mm/sec CNT100;
   1:  PR[91,1] = PR[90,1] + -21.989;
   1:  PR[91,2] = PR[90,2] + 17.991;
   1:L PR[91] R[100]mm/sec CNT100;
   1:  PR[91,1] = PR[90,1] + -22.965;
   1:  PR[91,2] = PR[90,2] + 17.838;
   1:L PR[91] R[100]mm/sec CNT100;
   1:  PR[91,1] = PR[90,1] + -24.888;
   1:  PR[91,2] = PR[90,2] + 17.399;
   1:L PR[91] R[100]mm/sec CNT100;
   1:  PR[91,1] = PR[90,1] + -28.152;
   1:  PR[91,2] = PR[90,2] + 16.155;
   1:L PR[91] R[100]mm/sec CNT100;
   1:  PR[91,1] = PR[90,1] + -29.200;
   1:  PR[91,2] = PR[90,2] + 15.588;
   1:L PR[91] R[100]mm/sec CNT100;
   1:  PR[91,1] = PR[90,1] + -31.401;
   1:  PR[91,2] = PR[90,2] + 14.164;
   1:L PR[91] R[100]mm/sec CNT100;
   1:  PR[91,1] = PR[90,1] + -32.104;
   1:  PR[91,2] = PR[90,2] + 13.648;
   1:L PR[91] R[100]mm/sec CNT100;
   1:  PR[91,1] = PR[90,1] + -34.845;
   1:  PR[91,2] = PR[90,2] + 10.906;
   1:L PR[91] R[100]mm/sec CNT100;
   1:  PR[91,1] = PR[90,1] + -35.095;
   1:  PR[91,2] = PR[90,2] + 10.581;
   1:L PR[91] R[100]mm/sec CNT100;
   1:  PR[91,1] = PR[90,1] + -37.010;
   1:  PR[91,2] = PR[90,2] + 7.525;
   1:L PR[91] R[100]mm/sec CNT100;
   1:  PR[91,1] = PR[90,1] + -37.122;
   1:  PR[91,2] = PR[90,2] + 7.324;
   1:L PR[91] R[100]mm/sec CNT100;
   1:  PR[91,1] = PR[90,1] + -38.479;
   1:  PR[91,2] = PR[90,2] + 3.580;
   1:L PR[91] R[100]mm/sec CNT100;
   1:  PR[91,1] = PR[90,1] + -38.481;
   1:  PR[91,2] = PR[90,2] + 3.571;
   1:L PR[91] R[100]mm/sec CNT100;
   1:  PR[91,1] = PR[90,1] + -38.923;
   1:  PR[91,2] = PR[90,2] + -0.420;
   1:L PR[91] R[100]mm/sec CNT100;
   1:  PR[91,1] = PR[90,1] + -38.481;
   1:  PR[91,2] = PR[90,2] + -4.305;
   1:L PR[91] R[100]mm/sec CNT100;
   1:  PR[91,1] = PR[90,1] + -38.471;
   1:  PR[91,2] = PR[90,2] + -4.449;
   1:L PR[91] R[100]mm/sec CNT100;
   1:  PR[91,1] = PR[90,1] + -37.122;
   1:  PR[91,2] = PR[90,2] + -8.172;
   1:L PR[91] R[100]mm/sec CNT100;
   1:  PR[91,1] = PR[90,1] + -37.009;
   1:  PR[91,2] = PR[90,2] + -8.374;
   1:L PR[91] R[100]mm/sec CNT100;
   1:  PR[91,1] = PR[90,1] + -35.093;
   1:  PR[91,2] = PR[90,2] + -11.430;
   1:L PR[91] R[100]mm/sec CNT100;
   1:  PR[91,1] = PR[90,1] + -34.844;
   1:  PR[91,2] = PR[90,2] + -11.755;
   1:L PR[91] R[100]mm/sec CNT100;
   1:  PR[91,1] = PR[90,1] + -32.102;
   1:  PR[91,2] = PR[90,2] + -14.497;
   1:L PR[91] R[100]mm/sec CNT100;
   1:  PR[91,1] = PR[90,1] + -31.400;
   1:  PR[91,2] = PR[90,2] + -15.013;
   1:L PR[91] R[100]mm/sec CNT100;
   1:  PR[91,1] = PR[90,1] + -29.198;
   1:  PR[91,2] = PR[90,2] + -16.436;
   1:L PR[91] R[100]mm/sec CNT100;
   1:  PR[91,1] = PR[90,1] + -28.151;
   1:  PR[91,2] = PR[90,2] + -17.003;
   1:L PR[91] R[100]mm/sec CNT100;
   1:  PR[91,1] = PR[90,1] + -24.886;
   1:  PR[91,2] = PR[90,2] + -18.247;
   1:L PR[91] R[100]mm/sec CNT100;
   1:  PR[91,1] = PR[90,1] + -22.964;
   1:  PR[91,2] = PR[90,2] + -18.685;
   1:L PR[91] R[100]mm/sec CNT100;
   1:  PR[91,1] = PR[90,1] + -21.988;
   1:  PR[91,2] = PR[90,2] + -18.839;
   1:L PR[91] R[100]mm/sec CNT100;
   1:  PR[91,1] = PR[90,1] + -19.723;
   1:  PR[91,2] = PR[90,2] + -19.045;
   1:L PR[91] R[100]mm/sec CNT100;
   1:  PR[91,1] = PR[90,1] + -16.789;
   1:  PR[91,2] = PR[90,2] + -18.929;
   1:L PR[91] R[100]mm/sec CNT100;
   1:  PR[91,1] = PR[90,1] + -14.122;
   1:  PR[91,2] = PR[90,2] + -18.482;
   1:L PR[91] R[100]mm/sec CNT100;
   1:  PR[91,1] = PR[90,1] + -11.224;
   1:  PR[91,2] = PR[90,2] + -17.578;
   1:L PR[91] R[100]mm/sec CNT100;
   1:  PR[91,1] = PR[90,1] + -9.110;
   1:  PR[91,2] = PR[90,2] + -16.584;
   1:L PR[91] R[100]mm/sec CNT100;
   1:  PR[91,1] = PR[90,1] + -8.388;
   1:  PR[91,2] = PR[90,2] + -16.178;
   1:L PR[91] R[100]mm/sec CNT100;
   1:  PR[91,1] = PR[90,1] + -6.498;
   1:  PR[91,2] = PR[90,2] + -14.943;
   1:L PR[91] R[100]mm/sec CNT100;
   1:  PR[91,1] = PR[90,1] + -6.170;
   1:  PR[91,2] = PR[90,2] + -14.670;
   1:L PR[91] R[100]mm/sec CNT100;
   1:  PR[91,1] = PR[90,1] + -4.786;
   1:  PR[91,2] = PR[90,2] + -13.454;
   1:L PR[91] R[100]mm/sec CNT100;
   1:  PR[91,1] = PR[90,1] + -4.304;
   1:  PR[91,2] = PR[90,2] + -12.977;
   1:L PR[91] R[100]mm/sec CNT100;
   1:  PR[91,1] = PR[90,1] + -3.676;
   1:  PR[91,2] = PR[90,2] + -12.233;
   1:L PR[91] R[100]mm/sec CNT100;
   1:  PR[91,1] = PR[90,1] + -3.535;
   1:  PR[91,2] = PR[90,2] + -11.986;
   1:L PR[91] R[100]mm/sec CNT100;
   1:  PR[91,1] = PR[90,1] + -3.371;
   1:  PR[91,2] = PR[90,2] + -11.872;
   1:L PR[91] R[100]mm/sec CNT100;
   1:  PR[91,1] = PR[90,1] + -2.970;
   1:  PR[91,2] = PR[90,2] + -11.397;
   1:L PR[91] R[100]mm/sec CNT100;
   1:  PR[91,1] = PR[90,1] + -2.672;
   1:  PR[91,2] = PR[90,2] + -11.384;
   1:L PR[91] R[100]mm/sec CNT100;
   1:  PR[91,1] = PR[90,1] + -2.231;
   1:  PR[91,2] = PR[90,2] + -11.086;
   1:L PR[91] R[100]mm/sec CNT100;
   1:  PR[91,1] = PR[90,1] + -0.857;
   1:  PR[91,2] = PR[90,2] + -10.783;
   1:L PR[91] R[100]mm/sec CNT100;
   1:  PR[91,1] = PR[90,1] + 0.328;
   1:L PR[91] R[100]mm/sec CNT100;
   1:  PR[91,1] = PR[90,1] + 1.745;
   1:  PR[91,2] = PR[90,2] + -11.078;
   1:L PR[91] R[100]mm/sec CNT100;
   1:  PR[91,1] = PR[90,1] + 2.410;
   1:  PR[91,2] = PR[90,2] + -11.526;
   1:L PR[91] R[100]mm/sec CNT100;
   1:  PR[91,1] = PR[90,1] + 2.700;
   1:  PR[91,2] = PR[90,2] + -11.796;
   1:L PR[91] R[100]mm/sec CNT100;
   1:  PR[91,1] = PR[90,1] + 2.914;
   1:  PR[91,2] = PR[90,2] + -11.946;
   1:L PR[91] R[100]mm/sec CNT100;
   1:  PR[91,1] = PR[90,1] + 3.821;
   1:  PR[91,2] = PR[90,2] + -12.971;
   1:L PR[91] R[100]mm/sec CNT100;
   1:  PR[91,1] = PR[90,1] + 4.324;
   1:  PR[91,2] = PR[90,2] + -13.471;
   1:L PR[91] R[100]mm/sec CNT100;
   1:  PR[91,1] = PR[90,1] + 5.706;
   1:  PR[91,2] = PR[90,2] + -14.685;
   1:L PR[91] R[100]mm/sec CNT100;
   1:  PR[91,1] = PR[90,1] + 6.033;
   1:  PR[91,2] = PR[90,2] + -14.958;
   1:L PR[91] R[100]mm/sec CNT100;
   1:  PR[91,1] = PR[90,1] + 7.906;
   1:  PR[91,2] = PR[90,2] + -16.179;
   1:L PR[91] R[100]mm/sec CNT100;
   1:  PR[91,1] = PR[90,1] + 8.627;
   1:  PR[91,2] = PR[90,2] + -16.585;
   1:L PR[91] R[100]mm/sec CNT100;
   1:  PR[91,1] = PR[90,1] + 10.732;
   1:  PR[91,2] = PR[90,2] + -17.572;
   1:L PR[91] R[100]mm/sec CNT100;
   1:  PR[91,1] = PR[90,1] + 13.637;
   1:  PR[91,2] = PR[90,2] + -18.479;
   1:L PR[91] R[100]mm/sec CNT100;
   1:  PR[91,1] = PR[90,1] + 16.305;
   1:  PR[91,2] = PR[90,2] + -18.929;
   1:L PR[91] R[100]mm/sec CNT100;
   1:  PR[91,1] = PR[90,1] + 19.230;
   1:  PR[91,2] = PR[90,2] + -19.046;
   1:L PR[91] R[100]mm/sec CNT100;
   1:  PR[91,1] = PR[90,1] + 21.490;
   1:  PR[91,2] = PR[90,2] + -18.842;
   1:L PR[91] R[100]mm/sec CNT100;
   1:  PR[91,1] = PR[90,1] + 22.461;
   1:  PR[91,2] = PR[90,2] + -18.689;
   1:L PR[91] R[100]mm/sec CNT100;
   1:  PR[91,1] = PR[90,1] + 24.392;
   1:  PR[91,2] = PR[90,2] + -18.249;
   1:L PR[91] R[100]mm/sec CNT100;
   1:  PR[91,1] = PR[90,1] + 27.667;
   1:  PR[91,2] = PR[90,2] + -17.005;
   1:L PR[91] R[100]mm/sec CNT100;
   1:  PR[91,1] = PR[90,1] + 28.712;
   1:  PR[91,2] = PR[90,2] + -16.443;
   1:L PR[91] R[100]mm/sec CNT100;
   1:  PR[91,1] = PR[90,1] + 30.913;
   1:  PR[91,2] = PR[90,2] + -15.020;
   1:L PR[91] R[100]mm/sec CNT100;
   1:  PR[91,1] = PR[90,1] + 31.610;
   1:  PR[91,2] = PR[90,2] + -14.511;
   1:L PR[91] R[100]mm/sec CNT100;
   1:  PR[91,1] = PR[90,1] + 34.355;
   1:  PR[91,2] = PR[90,2] + -11.758;
   1:L PR[91] R[100]mm/sec CNT100;
   1:  PR[91,1] = PR[90,1] + 34.611;
   1:  PR[91,2] = PR[90,2] + -11.425;
   1:L PR[91] R[100]mm/sec CNT100;
   1:  PR[91,1] = PR[90,1] + 36.529;
   1:  PR[91,2] = PR[90,2] + -8.371;
   1:L PR[91] R[100]mm/sec CNT100;
   1:  PR[91,1] = PR[90,1] + 36.643;
   1:  PR[91,2] = PR[90,2] + -8.168;
   1:L PR[91] R[100]mm/sec CNT100;
   1:  PR[91,1] = PR[90,1] + 37.999;
   1:  PR[91,2] = PR[90,2] + -4.445;
   1:L PR[91] R[100]mm/sec CNT100;
   1:  PR[91,1] = PR[90,1] + 38.000;
   1:  PR[91,2] = PR[90,2] + -4.440;
   1:L PR[91] R[100]mm/sec CNT100;
   1:  PR[91,1] = PR[90,1] + 38.443;
   1:  PR[91,2] = PR[90,2] + -0.427;
   1:L PR[91] R[100]mm/sec CNT100;
   1:  PR[91,1] = PR[90,1] + 38.001;
   1:  PR[91,2] = PR[90,2] + 3.471;
   1:L PR[91] R[100]mm/sec CNT100;
   1:  PR[91,1] = PR[90,1] + 37.991;
   1:  PR[91,2] = PR[90,2] + 3.622;
   1:L PR[91] R[100]mm/sec CNT100;
   1:  PR[91,1] = PR[90,1] + 36.740;
   1:  PR[91,2] = PR[90,2] + 7.085;
   1:L PR[91] R[100]mm/sec CNT100;
   1:  PR[91,1] = PR[90,1] + 36.657;
   1:  PR[91,2] = PR[90,2] + 7.297;
   1:L PR[91] R[100]mm/sec CNT100;
   1:  PR[91,1] = PR[90,1] + 36.529;
   1:  PR[91,2] = PR[90,2] + 7.524;
   1:L PR[91] R[100]mm/sec CNT100;
   1:  PR[91,1] = PR[90,1] + 34.611;
   1:  PR[91,2] = PR[90,2] + 10.578;
   1:L PR[91] R[100]mm/sec CNT100;
   1:  PR[91,1] = PR[90,1] + 34.352;
   1:  PR[91,2] = PR[90,2] + 10.915;
   1:L PR[91] R[100]mm/sec CNT100;
   1:  PR[91,1] = PR[90,1] + 32.141;
   1:  PR[91,2] = PR[90,2] + 13.147;
   1:L PR[91] R[100]mm/sec CNT100;
   1:  PR[91,1] = PR[90,1] + 31.622;
   1:  PR[91,2] = PR[90,2] + 13.655;
   1:L PR[91] R[100]mm/sec CNT100;
   1:  PR[91,1] = PR[90,1] + 30.913;
   1:  PR[91,2] = PR[90,2] + 14.173;
   1:L PR[91] R[100]mm/sec CNT100;
   1:  PR[91,1] = PR[90,1] + 28.712;
   1:  PR[91,2] = PR[90,2] + 15.596;
   1:L PR[91] R[100]mm/sec CNT100;
   1:  PR[91,1] = PR[90,1] + 27.666;
   1:  PR[91,2] = PR[90,2] + 16.158;
   1:L PR[91] R[100]mm/sec CNT100;
   1:  PR[91,1] = PR[90,1] + 24.392;
   1:  PR[91,2] = PR[90,2] + 17.402;
   1:L PR[91] R[100]mm/sec CNT100;
   1:  PR[91,1] = PR[90,1] + 22.461;
   1:  PR[91,2] = PR[90,2] + 17.842;
   1:L PR[91] R[100]mm/sec CNT100;
   1:  PR[91,1] = PR[90,1] + 21.490;
   1:  PR[91,2] = PR[90,2] + 17.995;
   1:L PR[91] R[100]mm/sec CNT100;
   1:  PR[91,1] = PR[90,1] + 19.230;
   1:  PR[91,2] = PR[90,2] + 18.198;
   1:L PR[91] R[100]mm/sec CNT100;
   1:  PR[91,1] = PR[90,1] + 16.305;
   1:  PR[91,2] = PR[90,2] + 18.082;
   1:L PR[91] R[100]mm/sec CNT100;
   1:  PR[91,1] = PR[90,1] + 13.637;
   1:  PR[91,2] = PR[90,2] + 17.632;
   1:L PR[91] R[100]mm/sec CNT100;
   1:  PR[91,1] = PR[90,1] + 10.732;
   1:  PR[91,2] = PR[90,2] + 16.725;
   1:L PR[91] R[100]mm/sec CNT100;
   1:  PR[91,1] = PR[90,1] + 8.627;
   1:  PR[91,2] = PR[90,2] + 15.737;
   1:L PR[91] R[100]mm/sec CNT100;
   1:  PR[91,1] = PR[90,1] + 7.906;
   1:  PR[91,2] = PR[90,2] + 15.332;
   1:L PR[91] R[100]mm/sec CNT100;
   1:  PR[91,1] = PR[90,1] + 6.035;
   1:  PR[91,2] = PR[90,2] + 14.112;
   1:L PR[91] R[100]mm/sec CNT100;
   1:  PR[91,1] = PR[90,1] + 5.707;
   1:  PR[91,2] = PR[90,2] + 13.838;
   1:L PR[91] R[100]mm/sec CNT100;
   1:  PR[91,1] = PR[90,1] + 4.325;
   1:  PR[91,2] = PR[90,2] + 12.624;
   1:L PR[91] R[100]mm/sec CNT100;
   1:  PR[91,1] = PR[90,1] + 3.837;
   1:  PR[91,2] = PR[90,2] + 12.139;
   1:L PR[91] R[100]mm/sec CNT100;
   1:  PR[91,1] = PR[90,1] + 2.876;
   1:  PR[91,2] = PR[90,2] + 11.011;
   1:L PR[91] R[100]mm/sec CNT100;
   1:  PR[91,1] = PR[90,1] + 2.275;
   1:  PR[91,2] = PR[90,2] + 10.588;
   1:L PR[91] R[100]mm/sec CNT100;
   1:  PR[91,1] = PR[90,1] + 1.758;
   1:  PR[91,2] = PR[90,2] + 10.239;
   1:L PR[91] R[100]mm/sec CNT100;
   1:  PR[91,1] = PR[90,1] + 0.383;
   1:  PR[91,2] = PR[90,2] + 9.936;
   1:L PR[91] R[100]mm/sec CNT100;
   1:  PR[91] = PR[90];
   1:  PR[91,1] = PR[90,1] + -0.632;
   1:  PR[91,2] = PR[90,2] + 10.480;
   1:  PR[91,3] = PR[90,3] + 27.495;
   1:L PR[91] R[100]mm/sec CNT100;
   1:  PR[91,1] = PR[90,1] + -2.147;
   1:  PR[91,2] = PR[90,2] + 10.793;
   1:L PR[91] R[100]mm/sec CNT100;
   1:  PR[91,1] = PR[90,1] + -2.711;
   1:  PR[91,2] = PR[90,2] + 11.275;
   1:L PR[91] R[100]mm/sec CNT100;
   1:  PR[91,1] = PR[90,1] + -3.186;
   1:  PR[91,2] = PR[90,2] + 11.606;
   1:L PR[91] R[100]mm/sec CNT100;
   1:  PR[91,1] = PR[90,1] + -3.671;
   1:  PR[91,2] = PR[90,2] + 12.152;
   1:L PR[91] R[100]mm/sec CNT100;
   1:  PR[91,1] = PR[90,1] + -4.391;
   1:  PR[91,2] = PR[90,2] + 12.865;
   1:L PR[91] R[100]mm/sec CNT100;
   1:  PR[91,1] = PR[90,1] + -5.462;
   1:  PR[91,2] = PR[90,2] + 13.806;
   1:L PR[91] R[100]mm/sec CNT100;
   1:  PR[91,1] = PR[90,1] + -5.984;
   1:  PR[91,2] = PR[90,2] + 14.240;
   1:L PR[91] R[100]mm/sec CNT100;
   1:  PR[91,1] = PR[90,1] + -7.604;
   1:  PR[91,2] = PR[90,2] + 15.299;
   1:L PR[91] R[100]mm/sec CNT100;
   1:  PR[91,1] = PR[90,1] + -8.784;
   1:  PR[91,2] = PR[90,2] + 15.963;
   1:L PR[91] R[100]mm/sec CNT100;
   1:  PR[91,1] = PR[90,1] + -10.612;
   1:  PR[91,2] = PR[90,2] + 16.822;
   1:L PR[91] R[100]mm/sec CNT100;
   1:  PR[91,1] = PR[90,1] + -13.712;
   1:  PR[91,2] = PR[90,2] + 17.785;
   1:L PR[91] R[100]mm/sec CNT100;
   1:  PR[91,1] = PR[90,1] + -16.095;
   1:  PR[91,2] = PR[90,2] + 18.184;
   1:L PR[91] R[100]mm/sec CNT100;
   1:  PR[91,1] = PR[90,1] + -16.588;
   1:  PR[91,2] = PR[90,2] + 18.223;
   1:L PR[91] R[100]mm/sec CNT100;
   1:  PR[91,1] = PR[90,1] + -19.160;
   1:  PR[91,2] = PR[90,2] + 18.310;
   1:L PR[91] R[100]mm/sec CNT100;
   1:  PR[91,1] = PR[90,1] + -22.024;
   1:  PR[91,2] = PR[90,2] + 18.025;
   1:L PR[91] R[100]mm/sec CNT100;
   1:  PR[91,1] = PR[90,1] + -24.647;
   1:  PR[91,2] = PR[90,2] + 17.426;
   1:L PR[91] R[100]mm/sec CNT100;
   1:  PR[91,1] = PR[90,1] + -27.563;
   1:  PR[91,2] = PR[90,2] + 16.314;
   1:L PR[91] R[100]mm/sec CNT100;
   1:  PR[91,1] = PR[90,1] + -29.196;
   1:  PR[91,2] = PR[90,2] + 15.430;
   1:L PR[91] R[100]mm/sec CNT100;
   1:  PR[91,1] = PR[90,1] + -30.525;
   1:  PR[91,2] = PR[90,2] + 14.570;
   1:L PR[91] R[100]mm/sec CNT100;
   1:  PR[91,1] = PR[90,1] + -31.802;
   1:  PR[91,2] = PR[90,2] + 13.632;
   1:L PR[91] R[100]mm/sec CNT100;
   1:  PR[91,1] = PR[90,1] + -34.305;
   1:  PR[91,2] = PR[90,2] + 11.139;
   1:L PR[91] R[100]mm/sec CNT100;
   1:  PR[91,1] = PR[90,1] + -34.931;
   1:  PR[91,2] = PR[90,2] + 10.324;
   1:L PR[91] R[100]mm/sec CNT100;
   1:  PR[91,1] = PR[90,1] + -36.336;
   1:  PR[91,2] = PR[90,2] + 8.081;
   1:L PR[91] R[100]mm/sec CNT100;
   1:  PR[91,1] = PR[90,1] + -36.771;
   1:  PR[91,2] = PR[90,2] + 7.304;
   1:L PR[91] R[100]mm/sec CNT100;
   1:  PR[91,1] = PR[90,1] + -37.748;
   1:  PR[91,2] = PR[90,2] + 4.594;
   1:L PR[91] R[100]mm/sec CNT100;
   1:  PR[91,1] = PR[90,1] + -38.050;
   1:  PR[91,2] = PR[90,2] + 3.807;
   1:L PR[91] R[100]mm/sec CNT100;
   1:  PR[91,1] = PR[90,1] + -38.174;
   1:  PR[91,2] = PR[90,2] + 3.255;
   1:L PR[91] R[100]mm/sec CNT100;
   1:  PR[91,1] = PR[90,1] + -38.520;
   1:  PR[91,2] = PR[90,2] + 0.191;
   1:L PR[91] R[100]mm/sec CNT100;
   1:  PR[91,1] = PR[90,1] + -38.559;
   1:  PR[91,2] = PR[90,2] + -0.370;
   1:L PR[91] R[100]mm/sec CNT100;
   1:  PR[91,1] = PR[90,1] + -38.212;
   1:  PR[91,2] = PR[90,2] + -3.417;
   1:L PR[91] R[100]mm/sec CNT100;
   1:  PR[91,1] = PR[90,1] + -38.162;
   1:  PR[91,2] = PR[90,2] + -4.155;
   1:L PR[91] R[100]mm/sec CNT100;
   1:  PR[91,1] = PR[90,1] + -38.044;
   1:  PR[91,2] = PR[90,2] + -4.680;
   1:L PR[91] R[100]mm/sec CNT100;
   1:  PR[91,1] = PR[90,1] + -37.082;
   1:  PR[91,2] = PR[90,2] + -7.356;
   1:L PR[91] R[100]mm/sec CNT100;
   1:  PR[91,1] = PR[90,1] + -36.783;
   1:  PR[91,2] = PR[90,2] + -8.129;
   1:L PR[91] R[100]mm/sec CNT100;
   1:  PR[91,1] = PR[90,1] + -36.336;
   1:  PR[91,2] = PR[90,2] + -8.929;
   1:L PR[91] R[100]mm/sec CNT100;
   1:  PR[91,1] = PR[90,1] + -34.930;
   1:  PR[91,2] = PR[90,2] + -11.172;
   1:L PR[91] R[100]mm/sec CNT100;
   1:  PR[91,1] = PR[90,1] + -34.301;
   1:  PR[91,2] = PR[90,2] + -11.992;
   1:L PR[91] R[100]mm/sec CNT100;
   1:  PR[91,1] = PR[90,1] + -32.741;
   1:  PR[91,2] = PR[90,2] + -13.561;
   1:L PR[91] R[100]mm/sec CNT100;
   1:  PR[91,1] = PR[90,1] + -31.809;
   1:  PR[91,2] = PR[90,2] + -14.475;
   1:L PR[91] R[100]mm/sec CNT100;
   1:  PR[91,1] = PR[90,1] + -30.524;
   1:  PR[91,2] = PR[90,2] + -15.418;
   1:L PR[91] R[100]mm/sec CNT100;
   1:  PR[91,1] = PR[90,1] + -29.195;
   1:  PR[91,2] = PR[90,2] + -16.277;
   1:L PR[91] R[100]mm/sec CNT100;
   1:  PR[91,1] = PR[90,1] + -27.562;
   1:  PR[91,2] = PR[90,2] + -17.161;
   1:L PR[91] R[100]mm/sec CNT100;
   1:  PR[91,1] = PR[90,1] + -24.647;
   1:  PR[91,2] = PR[90,2] + -18.273;
   1:L PR[91] R[100]mm/sec CNT100;
   1:  PR[91,1] = PR[90,1] + -22.021;
   1:  PR[91,2] = PR[90,2] + -18.872;
   1:L PR[91] R[100]mm/sec CNT100;
   1:  PR[91,1] = PR[90,1] + -19.275;
   1:  PR[91,2] = PR[90,2] + -19.134;
   1:L PR[91] R[100]mm/sec CNT100;
   1:  PR[91,1] = PR[90,1] + -19.118;
   1:  PR[91,2] = PR[90,2] + -19.155;
   1:L PR[91] R[100]mm/sec CNT100;
   1:  PR[91,1] = PR[90,1] + -16.588;
   1:  PR[91,2] = PR[90,2] + -19.071;
   1:L PR[91] R[100]mm/sec CNT100;
   1:  PR[91,1] = PR[90,1] + -16.095;
   1:  PR[91,2] = PR[90,2] + -19.031;
   1:L PR[91] R[100]mm/sec CNT100;
   1:  PR[91,1] = PR[90,1] + -13.712;
   1:  PR[91,2] = PR[90,2] + -18.632;
   1:L PR[91] R[100]mm/sec CNT100;
   1:  PR[91,1] = PR[90,1] + -10.612;
   1:  PR[91,2] = PR[90,2] + -17.669;
   1:L PR[91] R[100]mm/sec CNT100;
   1:  PR[91,1] = PR[90,1] + -8.784;
   1:  PR[91,2] = PR[90,2] + -16.810;
   1:L PR[91] R[100]mm/sec CNT100;
   1:  PR[91,1] = PR[90,1] + -7.603;
   1:  PR[91,2] = PR[90,2] + -16.146;
   1:L PR[91] R[100]mm/sec CNT100;
   1:  PR[91,1] = PR[90,1] + -5.994;
   1:  PR[91,2] = PR[90,2] + -15.095;
   1:L PR[91] R[100]mm/sec CNT100;
   1:  PR[91,1] = PR[90,1] + -5.460;
   1:  PR[91,2] = PR[90,2] + -14.651;
   1:L PR[91] R[100]mm/sec CNT100;
   1:  PR[91,1] = PR[90,1] + -4.391;
   1:  PR[91,2] = PR[90,2] + -13.712;
   1:L PR[91] R[100]mm/sec CNT100;
   1:  PR[91,1] = PR[90,1] + -3.692;
   1:  PR[91,2] = PR[90,2] + -13.020;
   1:L PR[91] R[100]mm/sec CNT100;
   1:  PR[91,1] = PR[90,1] + -3.520;
   1:  PR[91,2] = PR[90,2] + -12.816;
   1:L PR[91] R[100]mm/sec CNT100;
   1:  PR[91,1] = PR[90,1] + -3.370;
   1:  PR[91,2] = PR[90,2] + -12.554;
   1:L PR[91] R[100]mm/sec CNT100;
   1:  PR[91,1] = PR[90,1] + -3.195;
   1:  PR[91,2] = PR[90,2] + -12.432;
   1:L PR[91] R[100]mm/sec CNT100;
   1:  PR[91,1] = PR[90,1] + -2.752;
   1:  PR[91,2] = PR[90,2] + -11.907;
   1:L PR[91] R[100]mm/sec CNT100;
   1:  PR[91,1] = PR[90,1] + -2.425;
   1:  PR[91,2] = PR[90,2] + -11.893;
   1:L PR[91] R[100]mm/sec CNT100;
   1:  PR[91,1] = PR[90,1] + -2.014;
   1:  PR[91,2] = PR[90,2] + -11.616;
   1:L PR[91] R[100]mm/sec CNT100;
   1:  PR[91,1] = PR[90,1] + -0.659;
   1:  PR[91,2] = PR[90,2] + -11.327;
   1:L PR[91] R[100]mm/sec CNT100;
   1:  PR[91,1] = PR[90,1] + 0.158;
   1:L PR[91] R[100]mm/sec CNT100;
   1:  PR[91,1] = PR[90,1] + 1.673;
   1:  PR[91,2] = PR[90,2] + -11.641;
   1:L PR[91] R[100]mm/sec CNT100;
   1:  PR[91,1] = PR[90,1] + 2.241;
   1:  PR[91,2] = PR[90,2] + -12.125;
   1:L PR[91] R[100]mm/sec CNT100;
   1:  PR[91,1] = PR[90,1] + 2.716;
   1:  PR[91,2] = PR[90,2] + -12.457;
   1:L PR[91] R[100]mm/sec CNT100;
   1:  PR[91,1] = PR[90,1] + 3.204;
   1:  PR[91,2] = PR[90,2] + -13.009;
   1:L PR[91] R[100]mm/sec CNT100;
   1:  PR[91,1] = PR[90,1] + 3.925;
   1:  PR[91,2] = PR[90,2] + -13.726;
   1:L PR[91] R[100]mm/sec CNT100;
   1:  PR[91,1] = PR[90,1] + 4.993;
   1:  PR[91,2] = PR[90,2] + -14.664;
   1:L PR[91] R[100]mm/sec CNT100;
   1:  PR[91,1] = PR[90,1] + 5.514;
   1:  PR[91,2] = PR[90,2] + -15.099;
   1:L PR[91] R[100]mm/sec CNT100;
   1:  PR[91,1] = PR[90,1] + 7.120;
   1:  PR[91,2] = PR[90,2] + -16.147;
   1:L PR[91] R[100]mm/sec CNT100;
   1:  PR[91,1] = PR[90,1] + 8.300;
   1:  PR[91,2] = PR[90,2] + -16.810;
   1:L PR[91] R[100]mm/sec CNT100;
   1:  PR[91,1] = PR[90,1] + 10.120;
   1:  PR[91,2] = PR[90,2] + -17.664;
   1:L PR[91] R[100]mm/sec CNT100;
   1:  PR[91,1] = PR[90,1] + 13.227;
   1:  PR[91,2] = PR[90,2] + -18.629;
   1:L PR[91] R[100]mm/sec CNT100;
   1:  PR[91,1] = PR[90,1] + 15.611;
   1:  PR[91,2] = PR[90,2] + -19.031;
   1:L PR[91] R[100]mm/sec CNT100;
   1:  PR[91,1] = PR[90,1] + 16.104;
   1:  PR[91,2] = PR[90,2] + -19.071;
   1:L PR[91] R[100]mm/sec CNT100;
   1:  PR[91,1] = PR[90,1] + 18.665;
   1:  PR[91,2] = PR[90,2] + -19.158;
   1:L PR[91] R[100]mm/sec CNT100;
   1:  PR[91,1] = PR[90,1] + 21.515;
   1:  PR[91,2] = PR[90,2] + -18.877;
   1:L PR[91] R[100]mm/sec CNT100;
   1:  PR[91,1] = PR[90,1] + 24.144;
   1:  PR[91,2] = PR[90,2] + -18.278;
   1:L PR[91] R[100]mm/sec CNT100;
   1:  PR[91,1] = PR[90,1] + 27.072;
   1:  PR[91,2] = PR[90,2] + -17.166;
   1:L PR[91] R[100]mm/sec CNT100;
   1:  PR[91,1] = PR[90,1] + 28.703;
   1:  PR[91,2] = PR[90,2] + -16.288;
   1:L PR[91] R[100]mm/sec CNT100;
   1:  PR[91,1] = PR[90,1] + 30.029;
   1:  PR[91,2] = PR[90,2] + -15.431;
   1:L PR[91] R[100]mm/sec CNT100;
   1:  PR[91,1] = PR[90,1] + 31.293;
   1:  PR[91,2] = PR[90,2] + -14.507;
   1:L PR[91] R[100]mm/sec CNT100;
   1:  PR[91,1] = PR[90,1] + 32.815;
   1:  PR[91,2] = PR[90,2] + -12.973;
   1:L PR[91] R[100]mm/sec CNT100;
   1:  PR[91,1] = PR[90,1] + 33.810;
   1:  PR[91,2] = PR[90,2] + -11.996;
   1:L PR[91] R[100]mm/sec CNT100;
   1:  PR[91,1] = PR[90,1] + 34.442;
   1:  PR[91,2] = PR[90,2] + -11.175;
   1:L PR[91] R[100]mm/sec CNT100;
   1:  PR[91,1] = PR[90,1] + 35.849;
   1:  PR[91,2] = PR[90,2] + -8.934;
   1:L PR[91] R[100]mm/sec CNT100;
   1:  PR[91,1] = PR[90,1] + 36.289;
   1:  PR[91,2] = PR[90,2] + -8.155;
   1:L PR[91] R[100]mm/sec CNT100;
   1:  PR[91,1] = PR[90,1] + 37.266;
   1:  PR[91,2] = PR[90,2] + -5.458;
   1:L PR[91] R[100]mm/sec CNT100;
   1:  PR[91,1] = PR[90,1] + 37.567;
   1:  PR[91,2] = PR[90,2] + -4.683;
   1:L PR[91] R[100]mm/sec CNT100;
   1:  PR[91,1] = PR[90,1] + 37.691;
   1:  PR[91,2] = PR[90,2] + -4.139;
   1:L PR[91] R[100]mm/sec CNT100;
   1:  PR[91,1] = PR[90,1] + 38.037;
   1:  PR[91,2] = PR[90,2] + -1.064;
   1:L PR[91] R[100]mm/sec CNT100;
   1:  PR[91,1] = PR[90,1] + 38.079;
   1:  PR[91,2] = PR[90,2] + -0.475;
   1:L PR[91] R[100]mm/sec CNT100;
   1:  PR[91,1] = PR[90,1] + 37.733;
   1:  PR[91,2] = PR[90,2] + 2.579;
   1:L PR[91] R[100]mm/sec CNT100;
   1:  PR[91,1] = PR[90,1] + 37.679;
   1:  PR[91,2] = PR[90,2] + 3.342;
   1:L PR[91] R[100]mm/sec CNT100;
   1:  PR[91,1] = PR[90,1] + 37.561;
   1:  PR[91,2] = PR[90,2] + 3.864;
   1:L PR[91] R[100]mm/sec CNT100;
   1:  PR[91,1] = PR[90,1] + 36.599;
   1:  PR[91,2] = PR[90,2] + 6.526;
   1:L PR[91] R[100]mm/sec CNT100;
   1:  PR[91,1] = PR[90,1] + 36.304;
   1:  PR[91,2] = PR[90,2] + 7.281;
   1:L PR[91] R[100]mm/sec CNT100;
   1:  PR[91,1] = PR[90,1] + 35.849;
   1:  PR[91,2] = PR[90,2] + 8.087;
   1:L PR[91] R[100]mm/sec CNT100;
   1:  PR[91,1] = PR[90,1] + 34.442;
   1:  PR[91,2] = PR[90,2] + 10.328;
   1:L PR[91] R[100]mm/sec CNT100;
   1:  PR[91,1] = PR[90,1] + 33.799;
   1:  PR[91,2] = PR[90,2] + 11.163;
   1:L PR[91] R[100]mm/sec CNT100;
   1:  PR[91,1] = PR[90,1] + 32.241;
   1:  PR[91,2] = PR[90,2] + 12.737;
   1:L PR[91] R[100]mm/sec CNT100;
   1:  PR[91,1] = PR[90,1] + 31.308;
   1:  PR[91,2] = PR[90,2] + 13.649;
   1:L PR[91] R[100]mm/sec CNT100;
   1:  PR[91,1] = PR[90,1] + 30.029;
   1:  PR[91,2] = PR[90,2] + 14.584;
   1:L PR[91] R[100]mm/sec CNT100;
   1:  PR[91,1] = PR[90,1] + 28.703;
   1:  PR[91,2] = PR[90,2] + 15.441;
   1:L PR[91] R[100]mm/sec CNT100;
   1:  PR[91,1] = PR[90,1] + 27.071;
   1:  PR[91,2] = PR[90,2] + 16.319;
   1:L PR[91] R[100]mm/sec CNT100;
   1:  PR[91,1] = PR[90,1] + 24.144;
   1:  PR[91,2] = PR[90,2] + 17.431;
   1:L PR[91] R[100]mm/sec CNT100;
   1:  PR[91,1] = PR[90,1] + 21.520;
   1:  PR[91,2] = PR[90,2] + 18.029;
   1:L PR[91] R[100]mm/sec CNT100;
   1:  PR[91,1] = PR[90,1] + 18.781;
   1:  PR[91,2] = PR[90,2] + 18.287;
   1:L PR[91] R[100]mm/sec CNT100;
   1:  PR[91,1] = PR[90,1] + 18.622;
   1:  PR[91,2] = PR[90,2] + 18.309;
   1:L PR[91] R[100]mm/sec CNT100;
   1:  PR[91,1] = PR[90,1] + 16.104;
   1:  PR[91,2] = PR[90,2] + 18.223;
   1:L PR[91] R[100]mm/sec CNT100;
   1:  PR[91,1] = PR[90,1] + 15.611;
   1:  PR[91,2] = PR[90,2] + 18.184;
   1:L PR[91] R[100]mm/sec CNT100;
   1:  PR[91,1] = PR[90,1] + 13.227;
   1:  PR[91,2] = PR[90,2] + 17.782;
   1:L PR[91] R[100]mm/sec CNT100;
   1:  PR[91,1] = PR[90,1] + 10.121;
   1:  PR[91,2] = PR[90,2] + 16.816;
   1:L PR[91] R[100]mm/sec CNT100;
   1:  PR[91,1] = PR[90,1] + 8.300;
   1:  PR[91,2] = PR[90,2] + 15.963;
   1:L PR[91] R[100]mm/sec CNT100;
   1:  PR[91,1] = PR[90,1] + 7.120;
   1:  PR[91,2] = PR[90,2] + 15.300;
   1:L PR[91] R[100]mm/sec CNT100;
   1:  PR[91,1] = PR[90,1] + 5.527;
   1:  PR[91,2] = PR[90,2] + 14.261;
   1:L PR[91] R[100]mm/sec CNT100;
   1:  PR[91,1] = PR[90,1] + 4.994;
   1:  PR[91,2] = PR[90,2] + 13.818;
   1:L PR[91] R[100]mm/sec CNT100;
   1:  PR[91,1] = PR[90,1] + 3.926;
   1:  PR[91,2] = PR[90,2] + 12.879;
   1:L PR[91] R[100]mm/sec CNT100;
   1:  PR[91,1] = PR[90,1] + 3.220;
   1:  PR[91,2] = PR[90,2] + 12.178;
   1:L PR[91] R[100]mm/sec CNT100;
   1:  PR[91,1] = PR[90,1] + 2.710;
   1:  PR[91,2] = PR[90,2] + 11.579;
   1:L PR[91] R[100]mm/sec CNT100;
   1:  PR[91,1] = PR[90,1] + 2.003;
   1:  PR[91,2] = PR[90,2] + 11.081;
   1:L PR[91] R[100]mm/sec CNT100;
   1:  PR[91,1] = PR[90,1] + 1.541;
   1:  PR[91,2] = PR[90,2] + 10.769;
   1:L PR[91] R[100]mm/sec CNT100;
   1:  PR[91,1] = PR[90,1] + 0.184;
   1:  PR[91,2] = PR[90,2] + 10.480;
   1:L PR[91] R[100]mm/sec CNT100;
   1:  PR[91] = PR[90];
   1:  PR[91,1] = PR[90,1] + -1.329;
   1:  PR[91,2] = PR[90,2] + 11.091;
   1:  PR[91,3] = PR[90,3] + 28.795;
   1:L PR[91] R[100]mm/sec CNT100;
   1:  PR[91,1] = PR[90,1] + -2.893;
   1:  PR[91,2] = PR[90,2] + 12.031;
   1:L PR[91] R[100]mm/sec CNT100;
   1:  PR[91,1] = PR[90,1] + -3.996;
   1:  PR[91,2] = PR[90,2] + 13.124;
   1:L PR[91] R[100]mm/sec CNT100;
   1:  PR[91,1] = PR[90,1] + -4.753;
   1:  PR[91,2] = PR[90,2] + 13.789;
   1:L PR[91] R[100]mm/sec CNT100;
   1:  PR[91,1] = PR[90,1] + -5.468;
   1:  PR[91,2] = PR[90,2] + 14.384;
   1:L PR[91] R[100]mm/sec CNT100;
   1:  PR[91,1] = PR[90,1] + -6.819;
   1:  PR[91,2] = PR[90,2] + 15.267;
   1:L PR[91] R[100]mm/sec CNT100;
   1:  PR[91,1] = PR[90,1] + -8.458;
   1:  PR[91,2] = PR[90,2] + 16.189;
   1:L PR[91] R[100]mm/sec CNT100;
   1:  PR[91,1] = PR[90,1] + -9.999;
   1:  PR[91,2] = PR[90,2] + 16.913;
   1:L PR[91] R[100]mm/sec CNT100;
   1:  PR[91,1] = PR[90,1] + -13.302;
   1:  PR[91,2] = PR[90,2] + 17.934;
   1:L PR[91] R[100]mm/sec CNT100;
   1:  PR[91,1] = PR[90,1] + -15.353;
   1:  PR[91,2] = PR[90,2] + 18.278;
   1:L PR[91] R[100]mm/sec CNT100;
   1:  PR[91,1] = PR[90,1] + -16.390;
   1:  PR[91,2] = PR[90,2] + 18.361;
   1:L PR[91] R[100]mm/sec CNT100;
   1:  PR[91,1] = PR[90,1] + -18.641;
   1:  PR[91,2] = PR[90,2] + 18.436;
   1:L PR[91] R[100]mm/sec CNT100;
   1:  PR[91,1] = PR[90,1] + -21.248;
   1:  PR[91,2] = PR[90,2] + 18.177;
   1:L PR[91] R[100]mm/sec CNT100;
   1:  PR[91,1] = PR[90,1] + -21.668;
   1:  PR[91,2] = PR[90,2] + 18.121;
   1:L PR[91] R[100]mm/sec CNT100;
   1:  PR[91,1] = PR[90,1] + -24.233;
   1:  PR[91,2] = PR[90,2] + 17.514;
   1:L PR[91] R[100]mm/sec CNT100;
   1:  PR[91,1] = PR[90,1] + -26.975;
   1:  PR[91,2] = PR[90,2] + 16.471;
   1:L PR[91] R[100]mm/sec CNT100;
   1:  PR[91,1] = PR[90,1] + -29.193;
   1:  PR[91,2] = PR[90,2] + 15.271;
   1:L PR[91] R[100]mm/sec CNT100;
   1:  PR[91,1] = PR[90,1] + -29.649;
   1:  PR[91,2] = PR[90,2] + 14.976;
   1:L PR[91] R[100]mm/sec CNT100;
   1:  PR[91,1] = PR[90,1] + -31.501;
   1:  PR[91,2] = PR[90,2] + 13.616;
   1:L PR[91] R[100]mm/sec CNT100;
   1:  PR[91,1] = PR[90,1] + -33.766;
   1:  PR[91,2] = PR[90,2] + 11.372;
   1:L PR[91] R[100]mm/sec CNT100;
   1:  PR[91,1] = PR[90,1] + -34.767;
   1:  PR[91,2] = PR[90,2] + 10.067;
   1:L PR[91] R[100]mm/sec CNT100;
   1:  PR[91,1] = PR[90,1] + -35.663;
   1:  PR[91,2] = PR[90,2] + 8.637;
   1:L PR[91] R[100]mm/sec CNT100;
   1:  PR[91,1] = PR[90,1] + -36.421;
   1:  PR[91,2] = PR[90,2] + 7.282;
   1:L PR[91] R[100]mm/sec CNT100;
   1:  PR[91,1] = PR[90,1] + -37.078;
   1:  PR[91,2] = PR[90,2] + 5.460;
   1:L PR[91] R[100]mm/sec CNT100;
   1:  PR[91,1] = PR[90,1] + -37.617;
   1:  PR[91,2] = PR[90,2] + 4.057;
   1:L PR[91] R[100]mm/sec CNT100;
   1:  PR[91,1] = PR[90,1] + -37.866;
   1:  PR[91,2] = PR[90,2] + 2.941;
   1:L PR[91] R[100]mm/sec CNT100;
   1:  PR[91,1] = PR[90,1] + -38.110;
   1:  PR[91,2] = PR[90,2] + 0.785;
   1:L PR[91] R[100]mm/sec CNT100;
   1:  PR[91,1] = PR[90,1] + -38.189;
   1:  PR[91,2] = PR[90,2] + -0.370;
   1:L PR[91] R[100]mm/sec CNT100;
   1:  PR[91,1] = PR[90,1] + -37.943;
   1:  PR[91,2] = PR[90,2] + -2.528;
   1:L PR[91] R[100]mm/sec CNT100;
   1:  PR[91,1] = PR[90,1] + -37.854;
   1:  PR[91,2] = PR[90,2] + -3.841;
   1:L PR[91] R[100]mm/sec CNT100;
   1:  PR[91,1] = PR[90,1] + -37.611;
   1:  PR[91,2] = PR[90,2] + -4.930;
   1:L PR[91] R[100]mm/sec CNT100;
   1:  PR[91,1] = PR[90,1] + -36.944;
   1:  PR[91,2] = PR[90,2] + -6.782;
   1:L PR[91] R[100]mm/sec CNT100;
   1:  PR[91,1] = PR[90,1] + -36.433;
   1:  PR[91,2] = PR[90,2] + -8.107;
   1:L PR[91] R[100]mm/sec CNT100;
   1:  PR[91,1] = PR[90,1] + -35.663;
   1:  PR[91,2] = PR[90,2] + -9.485;
   1:L PR[91] R[100]mm/sec CNT100;
   1:  PR[91,1] = PR[90,1] + -34.766;
   1:  PR[91,2] = PR[90,2] + -10.915;
   1:L PR[91] R[100]mm/sec CNT100;
   1:  PR[91,1] = PR[90,1] + -33.760;
   1:  PR[91,2] = PR[90,2] + -12.227;
   1:L PR[91] R[100]mm/sec CNT100;
   1:  PR[91,1] = PR[90,1] + -32.851;
   1:  PR[91,2] = PR[90,2] + -13.141;
   1:L PR[91] R[100]mm/sec CNT100;
   1:  PR[91,1] = PR[90,1] + -31.506;
   1:  PR[91,2] = PR[90,2] + -14.460;
   1:L PR[91] R[100]mm/sec CNT100;
   1:  PR[91,1] = PR[90,1] + -29.648;
   1:  PR[91,2] = PR[90,2] + -15.824;
   1:L PR[91] R[100]mm/sec CNT100;
   1:  PR[91,1] = PR[90,1] + -29.193;
   1:  PR[91,2] = PR[90,2] + -16.118;
   1:L PR[91] R[100]mm/sec CNT100;
   1:  PR[91,1] = PR[90,1] + -26.975;
   1:  PR[91,2] = PR[90,2] + -17.319;
   1:L PR[91] R[100]mm/sec CNT100;
   1:  PR[91,1] = PR[90,1] + -24.233;
   1:  PR[91,2] = PR[90,2] + -18.361;
   1:L PR[91] R[100]mm/sec CNT100;
   1:  PR[91,1] = PR[90,1] + -21.712;
   1:  PR[91,2] = PR[90,2] + -18.958;
   1:L PR[91] R[100]mm/sec CNT100;
   1:  PR[91,1] = PR[90,1] + -19.273;
   1:  PR[91,2] = PR[90,2] + -19.191;
   1:L PR[91] R[100]mm/sec CNT100;
   1:  PR[91,1] = PR[90,1] + -18.598;
   1:  PR[91,2] = PR[90,2] + -19.282;
   1:L PR[91] R[100]mm/sec CNT100;
   1:  PR[91,1] = PR[90,1] + -16.390;
   1:  PR[91,2] = PR[90,2] + -19.208;
   1:L PR[91] R[100]mm/sec CNT100;
   1:  PR[91,1] = PR[90,1] + -15.353;
   1:  PR[91,2] = PR[90,2] + -19.125;
   1:L PR[91] R[100]mm/sec CNT100;
   1:  PR[91,1] = PR[90,1] + -13.308;
   1:  PR[91,2] = PR[90,2] + -18.782;
   1:L PR[91] R[100]mm/sec CNT100;
   1:  PR[91,1] = PR[90,1] + -11.475;
   1:  PR[91,2] = PR[90,2] + -18.206;
   1:L PR[91] R[100]mm/sec CNT100;
   1:  PR[91,1] = PR[90,1] + -9.992;
   1:  PR[91,2] = PR[90,2] + -17.757;
   1:L PR[91] R[100]mm/sec CNT100;
   1:  PR[91,1] = PR[90,1] + -8.458;
   1:  PR[91,2] = PR[90,2] + -17.036;
   1:L PR[91] R[100]mm/sec CNT100;
   1:  PR[91,1] = PR[90,1] + -6.818;
   1:  PR[91,2] = PR[90,2] + -16.114;
   1:L PR[91] R[100]mm/sec CNT100;
   1:  PR[91,1] = PR[90,1] + -5.481;
   1:  PR[91,2] = PR[90,2] + -15.241;
   1:L PR[91] R[100]mm/sec CNT100;
   1:  PR[91,1] = PR[90,1] + -4.750;
   1:  PR[91,2] = PR[90,2] + -14.634;
   1:L PR[91] R[100]mm/sec CNT100;
   1:  PR[91,1] = PR[90,1] + -3.995;
   1:  PR[91,2] = PR[90,2] + -13.970;
   1:L PR[91] R[100]mm/sec CNT100;
   1:  PR[91,1] = PR[90,1] + -2.893;
   1:  PR[91,2] = PR[90,2] + -12.878;
   1:L PR[91] R[100]mm/sec CNT100;
   1:  PR[91,1] = PR[90,1] + -1.326;
   1:  PR[91,2] = PR[90,2] + -11.937;
   1:L PR[91] R[100]mm/sec CNT100;
   1:  PR[91,1] = PR[90,1] + 0.863;
   1:  PR[91,2] = PR[90,2] + -11.942;
   1:L PR[91] R[100]mm/sec CNT100;
   1:  PR[91,1] = PR[90,1] + 2.423;
   1:  PR[91,2] = PR[90,2] + -12.884;
   1:L PR[91] R[100]mm/sec CNT100;
   1:  PR[91,1] = PR[90,1] + 3.526;
   1:  PR[91,2] = PR[90,2] + -13.981;
   1:L PR[91] R[100]mm/sec CNT100;
   1:  PR[91,1] = PR[90,1] + 4.280;
   1:  PR[91,2] = PR[90,2] + -14.643;
   1:L PR[91] R[100]mm/sec CNT100;
   1:  PR[91,1] = PR[90,1] + 4.995;
   1:  PR[91,2] = PR[90,2] + -15.240;
   1:L PR[91] R[100]mm/sec CNT100;
   1:  PR[91,1] = PR[90,1] + 6.335;
   1:  PR[91,2] = PR[90,2] + -16.115;
   1:L PR[91] R[100]mm/sec CNT100;
   1:  PR[91,1] = PR[90,1] + 7.974;
   1:  PR[91,2] = PR[90,2] + -17.036;
   1:L PR[91] R[100]mm/sec CNT100;
   1:  PR[91,1] = PR[90,1] + 9.509;
   1:  PR[91,2] = PR[90,2] + -17.755;
   1:L PR[91] R[100]mm/sec CNT100;
   1:  PR[91,1] = PR[90,1] + 12.817;
   1:  PR[91,2] = PR[90,2] + -18.779;
   1:L PR[91] R[100]mm/sec CNT100;
   1:  PR[91,1] = PR[90,1] + 14.869;
   1:  PR[91,2] = PR[90,2] + -19.125;
   1:L PR[91] R[100]mm/sec CNT100;
   1:  PR[91,1] = PR[90,1] + 15.906;
   1:  PR[91,2] = PR[90,2] + -19.208;
   1:L PR[91] R[100]mm/sec CNT100;
   1:  PR[91,1] = PR[90,1] + 18.147;
   1:  PR[91,2] = PR[90,2] + -19.284;
   1:L PR[91] R[100]mm/sec CNT100;
   1:  PR[91,1] = PR[90,1] + 20.740;
   1:  PR[91,2] = PR[90,2] + -19.029;
   1:L PR[91] R[100]mm/sec CNT100;
   1:  PR[91,1] = PR[90,1] + 21.163;
   1:  PR[91,2] = PR[90,2] + -18.973;
   1:L PR[91] R[100]mm/sec CNT100;
   1:  PR[91,1] = PR[90,1] + 23.725;
   1:  PR[91,2] = PR[90,2] + -18.367;
   1:L PR[91] R[100]mm/sec CNT100;
   1:  PR[91,1] = PR[90,1] + 26.478;
   1:  PR[91,2] = PR[90,2] + -17.326;
   1:L PR[91] R[100]mm/sec CNT100;
   1:  PR[91,1] = PR[90,1] + 28.693;
   1:  PR[91,2] = PR[90,2] + -16.134;
   1:L PR[91] R[100]mm/sec CNT100;
   1:  PR[91,1] = PR[90,1] + 29.145;
   1:  PR[91,2] = PR[90,2] + -15.842;
   1:L PR[91] R[100]mm/sec CNT100;
   1:  PR[91,1] = PR[90,1] + 30.979;
   1:  PR[91,2] = PR[90,2] + -14.501;
   1:L PR[91] R[100]mm/sec CNT100;
   1:  PR[91,1] = PR[90,1] + 31.737;
   1:  PR[91,2] = PR[90,2] + -13.737;
   1:L PR[91] R[100]mm/sec CNT100;
   1:  PR[91,1] = PR[90,1] + 33.258;
   1:  PR[91,2] = PR[90,2] + -12.244;
   1:L PR[91] R[100]mm/sec CNT100;
   1:  PR[91,1] = PR[90,1] + 34.273;
   1:  PR[91,2] = PR[90,2] + -10.926;
   1:L PR[91] R[100]mm/sec CNT100;
   1:  PR[91,1] = PR[90,1] + 35.170;
   1:  PR[91,2] = PR[90,2] + -9.497;
   1:L PR[91] R[100]mm/sec CNT100;
   1:  PR[91,1] = PR[90,1] + 35.936;
   1:  PR[91,2] = PR[90,2] + -8.140;
   1:L PR[91] R[100]mm/sec CNT100;
   1:  PR[91,1] = PR[90,1] + 36.592;
   1:  PR[91,2] = PR[90,2] + -6.327;
   1:L PR[91] R[100]mm/sec CNT100;
   1:  PR[91,1] = PR[90,1] + 37.130;
   1:  PR[91,2] = PR[90,2] + -4.946;
   1:L PR[91] R[100]mm/sec CNT100;
   1:  PR[91,1] = PR[90,1] + 37.380;
   1:  PR[91,2] = PR[90,2] + -3.840;
   1:L PR[91] R[100]mm/sec CNT100;
   1:  PR[91,1] = PR[90,1] + 37.624;
   1:  PR[91,2] = PR[90,2] + -1.677;
   1:L PR[91] R[100]mm/sec CNT100;
   1:  PR[91,1] = PR[90,1] + 37.709;
   1:  PR[91,2] = PR[90,2] + -0.475;
   1:L PR[91] R[100]mm/sec CNT100;
   1:  PR[91,1] = PR[90,1] + 37.464;
   1:  PR[91,2] = PR[90,2] + 1.688;
   1:L PR[91] R[100]mm/sec CNT100;
   1:  PR[91,1] = PR[90,1] + 37.369;
   1:  PR[91,2] = PR[90,2] + 3.043;
   1:L PR[91] R[100]mm/sec CNT100;
   1:  PR[91,1] = PR[90,1] + 37.123;
   1:  PR[91,2] = PR[90,2] + 4.127;
   1:L PR[91] R[100]mm/sec CNT100;
   1:  PR[91,1] = PR[90,1] + 36.458;
   1:  PR[91,2] = PR[90,2] + 5.968;
   1:L PR[91] R[100]mm/sec CNT100;
   1:  PR[91,1] = PR[90,1] + 35.951;
   1:  PR[91,2] = PR[90,2] + 7.266;
   1:L PR[91] R[100]mm/sec CNT100;
   1:  PR[91,1] = PR[90,1] + 35.170;
   1:  PR[91,2] = PR[90,2] + 8.650;
   1:L PR[91] R[100]mm/sec CNT100;
   1:  PR[91,1] = PR[90,1] + 34.273;
   1:  PR[91,2] = PR[90,2] + 10.078;
   1:L PR[91] R[100]mm/sec CNT100;
   1:  PR[91,1] = PR[90,1] + 33.247;
   1:  PR[91,2] = PR[90,2] + 11.411;
   1:L PR[91] R[100]mm/sec CNT100;
   1:  PR[91,1] = PR[90,1] + 32.341;
   1:  PR[91,2] = PR[90,2] + 12.327;
   1:L PR[91] R[100]mm/sec CNT100;
   1:  PR[91,1] = PR[90,1] + 30.994;
   1:  PR[91,2] = PR[90,2] + 13.643;
   1:L PR[91] R[100]mm/sec CNT100;
   1:  PR[91,1] = PR[90,1] + 29.145;
   1:  PR[91,2] = PR[90,2] + 14.995;
   1:L PR[91] R[100]mm/sec CNT100;
   1:  PR[91,1] = PR[90,1] + 28.693;
   1:  PR[91,2] = PR[90,2] + 15.287;
   1:L PR[91] R[100]mm/sec CNT100;
   1:  PR[91,1] = PR[90,1] + 26.477;
   1:  PR[91,2] = PR[90,2] + 16.479;
   1:L PR[91] R[100]mm/sec CNT100;
   1:  PR[91,1] = PR[90,1] + 23.817;
   1:  PR[91,2] = PR[90,2] + 17.489;
   1:L PR[91] R[100]mm/sec CNT100;
   1:  PR[91,1] = PR[90,1] + 23.745;
   1:  PR[91,2] = PR[90,2] + 17.515;
   1:L PR[91] R[100]mm/sec CNT100;
   1:  PR[91,1] = PR[90,1] + 21.207;
   1:  PR[91,2] = PR[90,2] + 18.115;
   1:L PR[91] R[100]mm/sec CNT100;
   1:  PR[91,1] = PR[90,1] + 18.781;
   1:  PR[91,2] = PR[90,2] + 18.344;
   1:L PR[91] R[100]mm/sec CNT100;
   1:  PR[91,1] = PR[90,1] + 18.104;
   1:  PR[91,2] = PR[90,2] + 18.436;
   1:L PR[91] R[100]mm/sec CNT100;
   1:  PR[91,1] = PR[90,1] + 15.906;
   1:  PR[91,2] = PR[90,2] + 18.361;
   1:L PR[91] R[100]mm/sec CNT100;
   1:  PR[91,1] = PR[90,1] + 14.869;
   1:  PR[91,2] = PR[90,2] + 18.277;
   1:L PR[91] R[100]mm/sec CNT100;
   1:  PR[91,1] = PR[90,1] + 12.823;
   1:  PR[91,2] = PR[90,2] + 17.932;
   1:L PR[91] R[100]mm/sec CNT100;
   1:  PR[91,1] = PR[90,1] + 10.987;
   1:  PR[91,2] = PR[90,2] + 17.354;
   1:L PR[91] R[100]mm/sec CNT100;
   1:  PR[91,1] = PR[90,1] + 9.502;
   1:  PR[91,2] = PR[90,2] + 16.905;
   1:L PR[91] R[100]mm/sec CNT100;
   1:  PR[91,1] = PR[90,1] + 7.974;
   1:  PR[91,2] = PR[90,2] + 16.188;
   1:L PR[91] R[100]mm/sec CNT100;
   1:  PR[91,1] = PR[90,1] + 6.335;
   1:  PR[91,2] = PR[90,2] + 15.268;
   1:L PR[91] R[100]mm/sec CNT100;
   1:  PR[91,1] = PR[90,1] + 5.012;
   1:  PR[91,2] = PR[90,2] + 14.405;
   1:L PR[91] R[100]mm/sec CNT100;
   1:  PR[91,1] = PR[90,1] + 4.281;
   1:  PR[91,2] = PR[90,2] + 13.797;
   1:L PR[91] R[100]mm/sec CNT100;
   1:  PR[91,1] = PR[90,1] + 3.527;
   1:  PR[91,2] = PR[90,2] + 13.134;
   1:L PR[91] R[100]mm/sec CNT100;
   1:  PR[91,1] = PR[90,1] + 2.406;
   1:  PR[91,2] = PR[90,2] + 12.021;
   1:L PR[91] R[100]mm/sec CNT100;
   1:  PR[91,1] = PR[90,1] + 0.853;
   1:  PR[91,2] = PR[90,2] + 11.093;
   1:L PR[91] R[100]mm/sec CNT100;
   1:  PR[91] = PR[90];
   1:  PR[91,1] = PR[90,1] + -1.152;
   1:  PR[91,2] = PR[90,2] + 11.679;
   1:  PR[91,3] = PR[90,3] + 30.095;
   1:L PR[91] R[100]mm/sec CNT100;
   1:  PR[91,1] = PR[90,1] + -2.078;
   1:  PR[91,2] = PR[90,2] + 12.116;
   1:L PR[91] R[100]mm/sec CNT100;
   1:  PR[91,1] = PR[90,1] + -2.317;
   1:  PR[91,2] = PR[90,2] + 12.320;
   1:L PR[91] R[100]mm/sec CNT100;
   1:  PR[91,1] = PR[90,1] + -2.854;
   1:  PR[91,2] = PR[90,2] + 12.643;
   1:L PR[91] R[100]mm/sec CNT100;
   1:  PR[91,1] = PR[90,1] + -3.601;
   1:  PR[91,2] = PR[90,2] + 13.382;
   1:L PR[91] R[100]mm/sec CNT100;
   1:  PR[91,1] = PR[90,1] + -4.044;
   1:  PR[91,2] = PR[90,2] + 13.771;
   1:L PR[91] R[100]mm/sec CNT100;
   1:  PR[91,1] = PR[90,1] + -4.952;
   1:  PR[91,2] = PR[90,2] + 14.527;
   1:L PR[91] R[100]mm/sec CNT100;
   1:  PR[91,1] = PR[90,1] + -6.034;
   1:  PR[91,2] = PR[90,2] + 15.235;
   1:L PR[91] R[100]mm/sec CNT100;
   1:  PR[91,1] = PR[90,1] + -8.132;
   1:  PR[91,2] = PR[90,2] + 16.415;
   1:L PR[91] R[100]mm/sec CNT100;
   1:  PR[91,1] = PR[90,1] + -9.387;
   1:  PR[91,2] = PR[90,2] + 17.005;
   1:L PR[91] R[100]mm/sec CNT100;
   1:  PR[91,1] = PR[90,1] + -12.892;
   1:  PR[91,2] = PR[90,2] + 18.084;
   1:L PR[91] R[100]mm/sec CNT100;
   1:  PR[91,1] = PR[90,1] + -14.611;
   1:  PR[91,2] = PR[90,2] + 18.372;
   1:L PR[91] R[100]mm/sec CNT100;
   1:  PR[91,1] = PR[90,1] + -16.191;
   1:  PR[91,2] = PR[90,2] + 18.498;
   1:L PR[91] R[100]mm/sec CNT100;
   1:  PR[91,1] = PR[90,1] + -18.121;
   1:  PR[91,2] = PR[90,2] + 18.563;
   1:L PR[91] R[100]mm/sec CNT100;
   1:  PR[91,1] = PR[90,1] + -20.363;
   1:  PR[91,2] = PR[90,2] + 18.340;
   1:L PR[91] R[100]mm/sec CNT100;
   1:  PR[91,1] = PR[90,1] + -21.363;
   1:  PR[91,2] = PR[90,2] + 18.207;
   1:L PR[91] R[100]mm/sec CNT100;
   1:  PR[91,1] = PR[90,1] + -23.594;
   1:  PR[91,2] = PR[90,2] + 17.678;
   1:L PR[91] R[100]mm/sec CNT100;
   1:  PR[91,1] = PR[90,1] + -26.525;
   1:  PR[91,2] = PR[90,2] + 16.575;
   1:L PR[91] R[100]mm/sec CNT100;
   1:  PR[91,1] = PR[90,1] + -28.965;
   1:  PR[91,2] = PR[90,2] + 15.243;
   1:L PR[91] R[100]mm/sec CNT100;
   1:  PR[91,1] = PR[90,1] + -28.988;
   1:  PR[91,2] = PR[90,2] + 15.228;
   1:L PR[91] R[100]mm/sec CNT100;
   1:  PR[91,1] = PR[90,1] + -31.200;
   1:  PR[91,2] = PR[90,2] + 13.600;
   1:L PR[91] R[100]mm/sec CNT100;
   1:  PR[91,1] = PR[90,1] + -33.227;
   1:  PR[91,2] = PR[90,2] + 11.604;
   1:L PR[91] R[100]mm/sec CNT100;
   1:  PR[91,1] = PR[90,1] + -34.603;
   1:  PR[91,2] = PR[90,2] + 9.811;
   1:L PR[91] R[100]mm/sec CNT100;
   1:  PR[91,1] = PR[90,1] + -34.990;
   1:  PR[91,2] = PR[90,2] + 9.193;
   1:L PR[91] R[100]mm/sec CNT100;
   1:  PR[91,1] = PR[90,1] + -36.070;
   1:  PR[91,2] = PR[90,2] + 7.261;
   1:L PR[91] R[100]mm/sec CNT100;
   1:  PR[91,1] = PR[90,1] + -36.407;
   1:  PR[91,2] = PR[90,2] + 6.326;
   1:L PR[91] R[100]mm/sec CNT100;
   1:  PR[91,1] = PR[90,1] + -37.183;
   1:  PR[91,2] = PR[90,2] + 4.307;
   1:L PR[91] R[100]mm/sec CNT100;
   1:  PR[91,1] = PR[90,1] + -37.558;
   1:  PR[91,2] = PR[90,2] + 2.627;
   1:L PR[91] R[100]mm/sec CNT100;
   1:  PR[91,1] = PR[90,1] + -37.699;
   1:  PR[91,2] = PR[90,2] + 1.379;
   1:L PR[91] R[100]mm/sec CNT100;
   1:  PR[91,1] = PR[90,1] + -37.819;
   1:  PR[91,2] = PR[90,2] + -0.370;
   1:L PR[91] R[100]mm/sec CNT100;
   1:  PR[91,1] = PR[90,1] + -37.675;
   1:  PR[91,2] = PR[90,2] + -1.640;
   1:L PR[91] R[100]mm/sec CNT100;
   1:  PR[91,1] = PR[90,1] + -37.546;
   1:  PR[91,2] = PR[90,2] + -3.527;
   1:L PR[91] R[100]mm/sec CNT100;
   1:  PR[91,1] = PR[90,1] + -37.177;
   1:  PR[91,2] = PR[90,2] + -5.179;
   1:L PR[91] R[100]mm/sec CNT100;
   1:  PR[91,1] = PR[90,1] + -36.807;
   1:  PR[91,2] = PR[90,2] + -6.207;
   1:L PR[91] R[100]mm/sec CNT100;
   1:  PR[91,1] = PR[90,1] + -36.083;
   1:  PR[91,2] = PR[90,2] + -8.085;
   1:L PR[91] R[100]mm/sec CNT100;
   1:  PR[91,1] = PR[90,1] + -34.990;
   1:  PR[91,2] = PR[90,2] + -10.041;
   1:L PR[91] R[100]mm/sec CNT100;
   1:  PR[91,1] = PR[90,1] + -34.603;
   1:  PR[91,2] = PR[90,2] + -10.658;
   1:L PR[91] R[100]mm/sec CNT100;
   1:  PR[91,1] = PR[90,1] + -33.219;
   1:  PR[91,2] = PR[90,2] + -12.462;
   1:L PR[91] R[100]mm/sec CNT100;
   1:  PR[91,1] = PR[90,1] + -32.959;
   1:  PR[91,2] = PR[90,2] + -12.723;
   1:L PR[91] R[100]mm/sec CNT100;
   1:  PR[91,1] = PR[90,1] + -31.202;
   1:  PR[91,2] = PR[90,2] + -14.445;
   1:L PR[91] R[100]mm/sec CNT100;
   1:  PR[91,1] = PR[90,1] + -28.988;
   1:  PR[91,2] = PR[90,2] + -16.075;
   1:L PR[91] R[100]mm/sec CNT100;
   1:  PR[91,1] = PR[90,1] + -28.965;
   1:  PR[91,2] = PR[90,2] + -16.090;
   1:L PR[91] R[100]mm/sec CNT100;
   1:  PR[91,1] = PR[90,1] + -26.520;
   1:  PR[91,2] = PR[90,2] + -17.425;
   1:L PR[91] R[100]mm/sec CNT100;
   1:  PR[91,1] = PR[90,1] + -24.204;
   1:  PR[91,2] = PR[90,2] + -18.309;
   1:L PR[91] R[100]mm/sec CNT100;
   1:  PR[91,1] = PR[90,1] + -23.612;
   1:  PR[91,2] = PR[90,2] + -18.521;
   1:L PR[91] R[100]mm/sec CNT100;
   1:  PR[91,1] = PR[90,1] + -21.406;
   1:  PR[91,2] = PR[90,2] + -19.044;
   1:L PR[91] R[100]mm/sec CNT100;
   1:  PR[91,1] = PR[90,1] + -19.272;
   1:  PR[91,2] = PR[90,2] + -19.248;
   1:L PR[91] R[100]mm/sec CNT100;
   1:  PR[91,1] = PR[90,1] + -18.079;
   1:  PR[91,2] = PR[90,2] + -19.409;
   1:L PR[91] R[100]mm/sec CNT100;
   1:  PR[91,1] = PR[90,1] + -16.191;
   1:  PR[91,2] = PR[90,2] + -19.346;
   1:L PR[91] R[100]mm/sec CNT100;
   1:  PR[91,1] = PR[90,1] + -14.611;
   1:  PR[91,2] = PR[90,2] + -19.219;
   1:L PR[91] R[100]mm/sec CNT100;
   1:  PR[91,1] = PR[90,1] + -12.899;
   1:  PR[91,2] = PR[90,2] + -18.932;
   1:L PR[91] R[100]mm/sec CNT100;
   1:  PR[91,1] = PR[90,1] + -11.352;
   1:  PR[91,2] = PR[90,2] + -18.445;
   1:L PR[91] R[100]mm/sec CNT100;
   1:  PR[91,1] = PR[90,1] + -9.381;
   1:  PR[91,2] = PR[90,2] + -17.849;
   1:L PR[91] R[100]mm/sec CNT100;
   1:  PR[91,1] = PR[90,1] + -8.131;
   1:  PR[91,2] = PR[90,2] + -17.262;
   1:L PR[91] R[100]mm/sec CNT100;
   1:  PR[91,1] = PR[90,1] + -6.032;
   1:  PR[91,2] = PR[90,2] + -16.081;
   1:L PR[91] R[100]mm/sec CNT100;
   1:  PR[91,1] = PR[90,1] + -4.969;
   1:  PR[91,2] = PR[90,2] + -15.387;
   1:L PR[91] R[100]mm/sec CNT100;
   1:  PR[91,1] = PR[90,1] + -4.040;
   1:  PR[91,2] = PR[90,2] + -14.616;
   1:L PR[91] R[100]mm/sec CNT100;
   1:  PR[91,1] = PR[90,1] + -3.599;
   1:  PR[91,2] = PR[90,2] + -14.228;
   1:L PR[91] R[100]mm/sec CNT100;
   1:  PR[91,1] = PR[90,1] + -2.869;
   1:  PR[91,2] = PR[90,2] + -13.505;
   1:L PR[91] R[100]mm/sec CNT100;
   1:  PR[91,1] = PR[90,1] + -0.990;
   1:  PR[91,2] = PR[90,2] + -12.331;
   1:L PR[91] R[100]mm/sec CNT100;
   1:  PR[91,1] = PR[90,1] + -0.090;
   1:  PR[91,2] = PR[90,2] + -12.582;
   1:L PR[91] R[100]mm/sec CNT100;
   1:  PR[91,1] = PR[90,1] + 1.018;
   1:  PR[91,2] = PR[90,2] + -12.583;
   1:L PR[91] R[100]mm/sec CNT100;
   1:  PR[91,1] = PR[90,1] + 1.759;
   1:  PR[91,2] = PR[90,2] + -13.119;
   1:L PR[91] R[100]mm/sec CNT100;
   1:  PR[91,1] = PR[90,1] + 2.382;
   1:  PR[91,2] = PR[90,2] + -13.495;
   1:L PR[91] R[100]mm/sec CNT100;
   1:  PR[91,1] = PR[90,1] + 3.127;
   1:  PR[91,2] = PR[90,2] + -14.236;
   1:L PR[91] R[100]mm/sec CNT100;
   1:  PR[91,1] = PR[90,1] + 3.567;
   1:  PR[91,2] = PR[90,2] + -14.622;
   1:L PR[91] R[100]mm/sec CNT100;
   1:  PR[91,1] = PR[90,1] + 4.476;
   1:  PR[91,2] = PR[90,2] + -15.380;
   1:L PR[91] R[100]mm/sec CNT100;
   1:  PR[91,1] = PR[90,1] + 5.550;
   1:  PR[91,2] = PR[90,2] + -16.083;
   1:L PR[91] R[100]mm/sec CNT100;
   1:  PR[91,1] = PR[90,1] + 7.647;
   1:  PR[91,2] = PR[90,2] + -17.261;
   1:L PR[91] R[100]mm/sec CNT100;
   1:  PR[91,1] = PR[90,1] + 8.897;
   1:  PR[91,2] = PR[90,2] + -17.847;
   1:L PR[91] R[100]mm/sec CNT100;
   1:  PR[91,1] = PR[90,1] + 12.408;
   1:  PR[91,2] = PR[90,2] + -18.928;
   1:L PR[91] R[100]mm/sec CNT100;
   1:  PR[91,1] = PR[90,1] + 14.127;
   1:  PR[91,2] = PR[90,2] + -19.218;
   1:L PR[91] R[100]mm/sec CNT100;
   1:  PR[91,1] = PR[90,1] + 15.707;
   1:  PR[91,2] = PR[90,2] + -19.346;
   1:L PR[91] R[100]mm/sec CNT100;
   1:  PR[91,1] = PR[90,1] + 17.629;
   1:  PR[91,2] = PR[90,2] + -19.411;
   1:L PR[91] R[100]mm/sec CNT100;
   1:  PR[91,1] = PR[90,1] + 19.858;
   1:  PR[91,2] = PR[90,2] + -19.192;
   1:L PR[91] R[100]mm/sec CNT100;
   1:  PR[91,1] = PR[90,1] + 20.860;
   1:  PR[91,2] = PR[90,2] + -19.058;
   1:L PR[91] R[100]mm/sec CNT100;
   1:  PR[91,1] = PR[90,1] + 23.089;
   1:  PR[91,2] = PR[90,2] + -18.531;
   1:L PR[91] R[100]mm/sec CNT100;
   1:  PR[91,1] = PR[90,1] + 26.029;
   1:  PR[91,2] = PR[90,2] + -17.429;
   1:L PR[91] R[100]mm/sec CNT100;
   1:  PR[91,1] = PR[90,1] + 28.458;
   1:  PR[91,2] = PR[90,2] + -16.110;
   1:L PR[91] R[100]mm/sec CNT100;
   1:  PR[91,1] = PR[90,1] + 28.484;
   1:  PR[91,2] = PR[90,2] + -16.094;
   1:L PR[91] R[100]mm/sec CNT100;
   1:  PR[91,1] = PR[90,1] + 30.676;
   1:  PR[91,2] = PR[90,2] + -14.487;
   1:L PR[91] R[100]mm/sec CNT100;
   1:  PR[91,1] = PR[90,1] + 32.705;
   1:  PR[91,2] = PR[90,2] + -12.493;
   1:L PR[91] R[100]mm/sec CNT100;
   1:  PR[91,1] = PR[90,1] + 34.104;
   1:  PR[91,2] = PR[90,2] + -10.676;
   1:L PR[91] R[100]mm/sec CNT100;
   1:  PR[91,1] = PR[90,1] + 34.490;
   1:  PR[91,2] = PR[90,2] + -10.061;
   1:L PR[91] R[100]mm/sec CNT100;
   1:  PR[91,1] = PR[90,1] + 35.583;
   1:  PR[91,2] = PR[90,2] + -8.125;
   1:L PR[91] R[100]mm/sec CNT100;
   1:  PR[91,1] = PR[90,1] + 35.919;
   1:  PR[91,2] = PR[90,2] + -7.196;
   1:L PR[91] R[100]mm/sec CNT100;
   1:  PR[91,1] = PR[90,1] + 36.692;
   1:  PR[91,2] = PR[90,2] + -5.208;
   1:L PR[91] R[100]mm/sec CNT100;
   1:  PR[91,1] = PR[90,1] + 37.070;
   1:  PR[91,2] = PR[90,2] + -3.542;
   1:L PR[91] R[100]mm/sec CNT100;
   1:  PR[91,1] = PR[90,1] + 37.211;
   1:  PR[91,2] = PR[90,2] + -2.291;
   1:L PR[91] R[100]mm/sec CNT100;
   1:  PR[91,1] = PR[90,1] + 37.339;
   1:  PR[91,2] = PR[90,2] + -0.475;
   1:L PR[91] R[100]mm/sec CNT100;
   1:  PR[91,1] = PR[90,1] + 37.195;
   1:  PR[91,2] = PR[90,2] + 0.796;
   1:L PR[91] R[100]mm/sec CNT100;
   1:  PR[91,1] = PR[90,1] + 37.059;
   1:  PR[91,2] = PR[90,2] + 2.744;
   1:L PR[91] R[100]mm/sec CNT100;
   1:  PR[91,1] = PR[90,1] + 36.686;
   1:  PR[91,2] = PR[90,2] + 4.390;
   1:L PR[91] R[100]mm/sec CNT100;
   1:  PR[91,1] = PR[90,1] + 36.318;
   1:  PR[91,2] = PR[90,2] + 5.410;
   1:L PR[91] R[100]mm/sec CNT100;
   1:  PR[91,1] = PR[90,1] + 35.598;
   1:  PR[91,2] = PR[90,2] + 7.251;
   1:L PR[91] R[100]mm/sec CNT100;
   1:  PR[91,1] = PR[90,1] + 34.490;
   1:  PR[91,2] = PR[90,2] + 9.214;
   1:L PR[91] R[100]mm/sec CNT100;
   1:  PR[91,1] = PR[90,1] + 34.104;
   1:  PR[91,2] = PR[90,2] + 9.829;
   1:L PR[91] R[100]mm/sec CNT100;
   1:  PR[91,1] = PR[90,1] + 32.705;
   1:  PR[91,2] = PR[90,2] + 11.646;
   1:L PR[91] R[100]mm/sec CNT100;
   1:  PR[91,1] = PR[90,1] + 30.676;
   1:  PR[91,2] = PR[90,2] + 13.640;
   1:L PR[91] R[100]mm/sec CNT100;
   1:  PR[91,1] = PR[90,1] + 28.484;
   1:  PR[91,2] = PR[90,2] + 15.247;
   1:L PR[91] R[100]mm/sec CNT100;
   1:  PR[91,1] = PR[90,1] + 28.458;
   1:  PR[91,2] = PR[90,2] + 15.263;
   1:L PR[91] R[100]mm/sec CNT100;
   1:  PR[91,1] = PR[90,1] + 26.025;
   1:  PR[91,2] = PR[90,2] + 16.584;
   1:L PR[91] R[100]mm/sec CNT100;
   1:  PR[91,1] = PR[90,1] + 23.702;
   1:  PR[91,2] = PR[90,2] + 17.466;
   1:L PR[91] R[100]mm/sec CNT100;
   1:  PR[91,1] = PR[90,1] + 23.106;
   1:  PR[91,2] = PR[90,2] + 17.680;
   1:L PR[91] R[100]mm/sec CNT100;
   1:  PR[91,1] = PR[90,1] + 20.904;
   1:  PR[91,2] = PR[90,2] + 18.201;
   1:L PR[91] R[100]mm/sec CNT100;
   1:  PR[91,1] = PR[90,1] + 18.780;
   1:  PR[91,2] = PR[90,2] + 18.401;
   1:L PR[91] R[100]mm/sec CNT100;
   1:  PR[91,1] = PR[90,1] + 17.585;
   1:  PR[91,2] = PR[90,2] + 18.562;
   1:L PR[91] R[100]mm/sec CNT100;
   1:  PR[91,1] = PR[90,1] + 15.707;
   1:  PR[91,2] = PR[90,2] + 18.498;
   1:L PR[91] R[100]mm/sec CNT100;
   1:  PR[91,1] = PR[90,1] + 14.127;
   1:  PR[91,2] = PR[90,2] + 18.371;
   1:L PR[91] R[100]mm/sec CNT100;
   1:  PR[91,1] = PR[90,1] + 12.415;
   1:  PR[91,2] = PR[90,2] + 18.082;
   1:L PR[91] R[100]mm/sec CNT100;
   1:  PR[91,1] = PR[90,1] + 10.865;
   1:  PR[91,2] = PR[90,2] + 17.594;
   1:L PR[91] R[100]mm/sec CNT100;
   1:  PR[91,1] = PR[90,1] + 8.892;
   1:  PR[91,2] = PR[90,2] + 16.997;
   1:L PR[91] R[100]mm/sec CNT100;
   1:  PR[91,1] = PR[90,1] + 7.647;
   1:  PR[91,2] = PR[90,2] + 16.414;
   1:L PR[91] R[100]mm/sec CNT100;
   1:  PR[91,1] = PR[90,1] + 5.549;
   1:  PR[91,2] = PR[90,2] + 15.235;
   1:L PR[91] R[100]mm/sec CNT100;
   1:  PR[91,1] = PR[90,1] + 4.497;
   1:  PR[91,2] = PR[90,2] + 14.549;
   1:L PR[91] R[100]mm/sec CNT100;
   1:  PR[91,1] = PR[90,1] + 3.569;
   1:  PR[91,2] = PR[90,2] + 13.777;
   1:L PR[91] R[100]mm/sec CNT100;
   1:  PR[91,1] = PR[90,1] + 3.122;
   1:  PR[91,2] = PR[90,2] + 13.384;
   1:L PR[91] R[100]mm/sec CNT100;
   1:  PR[91,1] = PR[90,1] + 2.282;
   1:  PR[91,2] = PR[90,2] + 12.561;
   1:L PR[91] R[100]mm/sec CNT100;
   1:  PR[91,1] = PR[90,1] + 1.325;
   1:  PR[91,2] = PR[90,2] + 11.987;
   1:L PR[91] R[100]mm/sec CNT100;
   1:  PR[91,1] = PR[90,1] + 0.592;
   1:  PR[91,2] = PR[90,2] + 11.681;
   1:L PR[91] R[100]mm/sec CNT100;
   1:  PR[91] = PR[90];
   1:  PR[91,1] = PR[90,1] + -1.097;
   1:  PR[91,2] = PR[90,2] + 12.268;
   1:  PR[91,3] = PR[90,3] + 31.395;
   1:L PR[91] R[100]mm/sec CNT100;
   1:  PR[91,1] = PR[90,1] + -2.168;
   1:  PR[91,2] = PR[90,2] + 12.764;
   1:L PR[91] R[100]mm/sec CNT100;
   1:  PR[91,1] = PR[90,1] + -2.559;
   1:  PR[91,2] = PR[90,2] + 13.100;
   1:L PR[91] R[100]mm/sec CNT100;
   1:  PR[91,1] = PR[90,1] + -2.788;
   1:  PR[91,2] = PR[90,2] + 13.238;
   1:L PR[91] R[100]mm/sec CNT100;
   1:  PR[91,1] = PR[90,1] + -3.364;
   1:  PR[91,2] = PR[90,2] + 13.778;
   1:L PR[91] R[100]mm/sec CNT100;
   1:  PR[91,1] = PR[90,1] + -4.437;
   1:  PR[91,2] = PR[90,2] + 14.671;
   1:L PR[91] R[100]mm/sec CNT100;
   1:  PR[91,1] = PR[90,1] + -5.250;
   1:  PR[91,2] = PR[90,2] + 15.204;
   1:L PR[91] R[100]mm/sec CNT100;
   1:  PR[91,1] = PR[90,1] + -7.805;
   1:  PR[91,2] = PR[90,2] + 16.641;
   1:L PR[91] R[100]mm/sec CNT100;
   1:  PR[91,1] = PR[90,1] + -8.775;
   1:  PR[91,2] = PR[90,2] + 17.096;
   1:L PR[91] R[100]mm/sec CNT100;
   1:  PR[91,1] = PR[90,1] + -12.483;
   1:  PR[91,2] = PR[90,2] + 18.233;
   1:L PR[91] R[100]mm/sec CNT100;
   1:  PR[91,1] = PR[90,1] + -13.869;
   1:  PR[91,2] = PR[90,2] + 18.466;
   1:L PR[91] R[100]mm/sec CNT100;
   1:  PR[91,1] = PR[90,1] + -15.993;
   1:  PR[91,2] = PR[90,2] + 18.636;
   1:L PR[91] R[100]mm/sec CNT100;
   1:  PR[91,1] = PR[90,1] + -17.601;
   1:  PR[91,2] = PR[90,2] + 18.690;
   1:L PR[91] R[100]mm/sec CNT100;
   1:  PR[91,1] = PR[90,1] + -19.477;
   1:  PR[91,2] = PR[90,2] + 18.503;
   1:L PR[91] R[100]mm/sec CNT100;
   1:  PR[91,1] = PR[90,1] + -21.057;
   1:  PR[91,2] = PR[90,2] + 18.293;
   1:L PR[91] R[100]mm/sec CNT100;
   1:  PR[91,1] = PR[90,1] + -22.948;
   1:  PR[91,2] = PR[90,2] + 17.845;
   1:L PR[91] R[100]mm/sec CNT100;
   1:  PR[91,1] = PR[90,1] + -25.185;
   1:  PR[91,2] = PR[90,2] + 16.996;
   1:L PR[91] R[100]mm/sec CNT100;
   1:  PR[91,1] = PR[90,1] + -26.115;
   1:  PR[91,2] = PR[90,2] + 16.661;
   1:L PR[91] R[100]mm/sec CNT100;
   1:  PR[91,1] = PR[90,1] + -28.214;
   1:  PR[91,2] = PR[90,2] + 15.515;
   1:L PR[91] R[100]mm/sec CNT100;
   1:  PR[91,1] = PR[90,1] + -28.738;
   1:  PR[91,2] = PR[90,2] + 15.189;
   1:L PR[91] R[100]mm/sec CNT100;
   1:  PR[91,1] = PR[90,1] + -30.710;
   1:  PR[91,2] = PR[90,2] + 13.734;
   1:L PR[91] R[100]mm/sec CNT100;
   1:  PR[91,1] = PR[90,1] + -32.764;
   1:  PR[91,2] = PR[90,2] + 11.736;
   1:L PR[91] R[100]mm/sec CNT100;
   1:  PR[91,1] = PR[90,1] + -34.378;
   1:  PR[91,2] = PR[90,2] + 9.633;
   1:L PR[91] R[100]mm/sec CNT100;
   1:  PR[91,1] = PR[90,1] + -35.732;
   1:  PR[91,2] = PR[90,2] + 7.218;
   1:L PR[91] R[100]mm/sec CNT100;
   1:  PR[91,1] = PR[90,1] + -36.749;
   1:  PR[91,2] = PR[90,2] + 4.558;
   1:L PR[91] R[100]mm/sec CNT100;
   1:  PR[91,1] = PR[90,1] + -37.250;
   1:  PR[91,2] = PR[90,2] + 2.313;
   1:L PR[91] R[100]mm/sec CNT100;
   1:  PR[91,1] = PR[90,1] + -37.289;
   1:  PR[91,2] = PR[90,2] + 1.972;
   1:L PR[91] R[100]mm/sec CNT100;
   1:  PR[91,1] = PR[90,1] + -37.450;
   1:  PR[91,2] = PR[90,2] + -0.370;
   1:L PR[91] R[100]mm/sec CNT100;
   1:  PR[91,1] = PR[90,1] + -37.406;
   1:  PR[91,2] = PR[90,2] + -0.751;
   1:L PR[91] R[100]mm/sec CNT100;
   1:  PR[91,1] = PR[90,1] + -37.239;
   1:  PR[91,2] = PR[90,2] + -3.213;
   1:L PR[91] R[100]mm/sec CNT100;
   1:  PR[91,1] = PR[90,1] + -36.749;
   1:  PR[91,2] = PR[90,2] + -5.406;
   1:L PR[91] R[100]mm/sec CNT100;
   1:  PR[91,1] = PR[90,1] + -35.732;
   1:  PR[91,2] = PR[90,2] + -8.065;
   1:L PR[91] R[100]mm/sec CNT100;
   1:  PR[91,1] = PR[90,1] + -34.378;
   1:  PR[91,2] = PR[90,2] + -10.480;
   1:L PR[91] R[100]mm/sec CNT100;
   1:  PR[91,1] = PR[90,1] + -32.764;
   1:  PR[91,2] = PR[90,2] + -12.583;
   1:L PR[91] R[100]mm/sec CNT100;
   1:  PR[91,1] = PR[90,1] + -30.710;
   1:  PR[91,2] = PR[90,2] + -14.582;
   1:L PR[91] R[100]mm/sec CNT100;
   1:  PR[91,1] = PR[90,1] + -28.738;
   1:  PR[91,2] = PR[90,2] + -16.036;
   1:L PR[91] R[100]mm/sec CNT100;
   1:  PR[91,1] = PR[90,1] + -28.213;
   1:  PR[91,2] = PR[90,2] + -16.363;
   1:L PR[91] R[100]mm/sec CNT100;
   1:  PR[91,1] = PR[90,1] + -26.095;
   1:  PR[91,2] = PR[90,2] + -17.520;
   1:L PR[91] R[100]mm/sec CNT100;
   1:  PR[91,1] = PR[90,1] + -24.087;
   1:  PR[91,2] = PR[90,2] + -18.286;
   1:L PR[91] R[100]mm/sec CNT100;
   1:  PR[91,1] = PR[90,1] + -22.969;
   1:  PR[91,2] = PR[90,2] + -18.687;
   1:L PR[91] R[100]mm/sec CNT100;
   1:  PR[91,1] = PR[90,1] + -21.100;
   1:  PR[91,2] = PR[90,2] + -19.130;
   1:L PR[91] R[100]mm/sec CNT100;
   1:  PR[91,1] = PR[90,1] + -19.270;
   1:  PR[91,2] = PR[90,2] + -19.305;
   1:L PR[91] R[100]mm/sec CNT100;
   1:  PR[91,1] = PR[90,1] + -17.559;
   1:  PR[91,2] = PR[90,2] + -19.535;
   1:L PR[91] R[100]mm/sec CNT100;
   1:  PR[91,1] = PR[90,1] + -15.993;
   1:  PR[91,2] = PR[90,2] + -19.483;
   1:L PR[91] R[100]mm/sec CNT100;
   1:  PR[91,1] = PR[90,1] + -13.869;
   1:  PR[91,2] = PR[90,2] + -19.313;
   1:L PR[91] R[100]mm/sec CNT100;
   1:  PR[91,1] = PR[90,1] + -12.491;
   1:  PR[91,2] = PR[90,2] + -19.082;
   1:L PR[91] R[100]mm/sec CNT100;
   1:  PR[91,1] = PR[90,1] + -11.230;
   1:  PR[91,2] = PR[90,2] + -18.685;
   1:L PR[91] R[100]mm/sec CNT100;
   1:  PR[91,1] = PR[90,1] + -8.770;
   1:  PR[91,2] = PR[90,2] + -17.941;
   1:L PR[91] R[100]mm/sec CNT100;
   1:  PR[91,1] = PR[90,1] + -7.805;
   1:  PR[91,2] = PR[90,2] + -17.488;
   1:L PR[91] R[100]mm/sec CNT100;
   1:  PR[91,1] = PR[90,1] + -5.247;
   1:  PR[91,2] = PR[90,2] + -16.049;
   1:L PR[91] R[100]mm/sec CNT100;
   1:  PR[91,1] = PR[90,1] + -4.456;
   1:  PR[91,2] = PR[90,2] + -15.533;
   1:L PR[91] R[100]mm/sec CNT100;
   1:  PR[91,1] = PR[90,1] + -3.361;
   1:  PR[91,2] = PR[90,2] + -14.622;
   1:L PR[91] R[100]mm/sec CNT100;
   1:  PR[91,1] = PR[90,1] + -2.818;
   1:  PR[91,2] = PR[90,2] + -14.113;
   1:L PR[91] R[100]mm/sec CNT100;
   1:  PR[91,1] = PR[90,1] + -0.965;
   1:  PR[91,2] = PR[90,2] + -12.913;
   1:L PR[91] R[100]mm/sec CNT100;
   1:  PR[91,1] = PR[90,1] + 0.151;
   1:  PR[91,2] = PR[90,2] + -13.224;
   1:L PR[91] R[100]mm/sec CNT100;
   1:  PR[91,1] = PR[90,1] + 1.066;
   1:  PR[91,2] = PR[90,2] + -13.225;
   1:L PR[91] R[100]mm/sec CNT100;
   1:  PR[91,1] = PR[90,1] + 1.997;
   1:  PR[91,2] = PR[90,2] + -13.899;
   1:L PR[91] R[100]mm/sec CNT100;
   1:  PR[91,1] = PR[90,1] + 2.312;
   1:  PR[91,2] = PR[90,2] + -14.089;
   1:L PR[91] R[100]mm/sec CNT100;
   1:  PR[91,1] = PR[90,1] + 2.885;
   1:  PR[91,2] = PR[90,2] + -14.628;
   1:L PR[91] R[100]mm/sec CNT100;
   1:  PR[91,1] = PR[90,1] + 3.958;
   1:  PR[91,2] = PR[90,2] + -15.522;
   1:L PR[91] R[100]mm/sec CNT100;
   1:  PR[91,1] = PR[90,1] + 4.765;
   1:  PR[91,2] = PR[90,2] + -16.051;
   1:L PR[91] R[100]mm/sec CNT100;
   1:  PR[91,1] = PR[90,1] + 7.321;
   1:  PR[91,2] = PR[90,2] + -17.487;
   1:L PR[91] R[100]mm/sec CNT100;
   1:  PR[91,1] = PR[90,1] + 8.286;
   1:  PR[91,2] = PR[90,2] + -17.939;
   1:L PR[91] R[100]mm/sec CNT100;
   1:  PR[91,1] = PR[90,1] + 11.998;
   1:  PR[91,2] = PR[90,2] + -19.078;
   1:L PR[91] R[100]mm/sec CNT100;
   1:  PR[91,1] = PR[90,1] + 13.385;
   1:  PR[91,2] = PR[90,2] + -19.312;
   1:L PR[91] R[100]mm/sec CNT100;
   1:  PR[91,1] = PR[90,1] + 15.509;
   1:  PR[91,2] = PR[90,2] + -19.483;
   1:L PR[91] R[100]mm/sec CNT100;
   1:  PR[91,1] = PR[90,1] + 17.110;
   1:  PR[91,2] = PR[90,2] + -19.537;
   1:L PR[91] R[100]mm/sec CNT100;
   1:  PR[91,1] = PR[90,1] + 18.976;
   1:  PR[91,2] = PR[90,2] + -19.354;
   1:L PR[91] R[100]mm/sec CNT100;
   1:  PR[91,1] = PR[90,1] + 20.557;
   1:  PR[91,2] = PR[90,2] + -19.144;
   1:L PR[91] R[100]mm/sec CNT100;
   1:  PR[91,1] = PR[90,1] + 22.446;
   1:  PR[91,2] = PR[90,2] + -18.697;
   1:L PR[91] R[100]mm/sec CNT100;
   1:  PR[91,1] = PR[90,1] + 24.688;
   1:  PR[91,2] = PR[90,2] + -17.851;
   1:L PR[91] R[100]mm/sec CNT100;
   1:  PR[91,1] = PR[90,1] + 25.621;
   1:  PR[91,2] = PR[90,2] + -17.515;
   1:L PR[91] R[100]mm/sec CNT100;
   1:  PR[91,1] = PR[90,1] + 27.710;
   1:  PR[91,2] = PR[90,2] + -16.381;
   1:L PR[91] R[100]mm/sec CNT100;
   1:  PR[91,1] = PR[90,1] + 28.236;
   1:  PR[91,2] = PR[90,2] + -16.053;
   1:L PR[91] R[100]mm/sec CNT100;
   1:  PR[91,1] = PR[90,1] + 30.188;
   1:  PR[91,2] = PR[90,2] + -14.621;
   1:L PR[91] R[100]mm/sec CNT100;
   1:  PR[91,1] = PR[90,1] + 32.240;
   1:  PR[91,2] = PR[90,2] + -12.628;
   1:L PR[91] R[100]mm/sec CNT100;
   1:  PR[91,1] = PR[90,1] + 33.874;
   1:  PR[91,2] = PR[90,2] + -10.505;
   1:L PR[91] R[100]mm/sec CNT100;
   1:  PR[91,1] = PR[90,1] + 35.243;
   1:  PR[91,2] = PR[90,2] + -8.085;
   1:L PR[91] R[100]mm/sec CNT100;
   1:  PR[91,1] = PR[90,1] + 36.255;
   1:  PR[91,2] = PR[90,2] + -5.473;
   1:L PR[91] R[100]mm/sec CNT100;
   1:  PR[91,1] = PR[90,1] + 36.760;
   1:  PR[91,2] = PR[90,2] + -3.243;
   1:L PR[91] R[100]mm/sec CNT100;
   1:  PR[91,1] = PR[90,1] + 36.798;
   1:  PR[91,2] = PR[90,2] + -2.904;
   1:L PR[91] R[100]mm/sec CNT100;
   1:  PR[91,1] = PR[90,1] + 36.970;
   1:  PR[91,2] = PR[90,2] + -0.475;
   1:L PR[91] R[100]mm/sec CNT100;
   1:  PR[91,1] = PR[90,1] + 36.927;
   1:  PR[91,2] = PR[90,2] + -0.096;
   1:L PR[91] R[100]mm/sec CNT100;
   1:  PR[91,1] = PR[90,1] + 36.749;
   1:  PR[91,2] = PR[90,2] + 2.446;
   1:L PR[91] R[100]mm/sec CNT100;
   1:  PR[91,1] = PR[90,1] + 36.255;
   1:  PR[91,2] = PR[90,2] + 4.626;
   1:L PR[91] R[100]mm/sec CNT100;
   1:  PR[91,1] = PR[90,1] + 35.243;
   1:  PR[91,2] = PR[90,2] + 7.238;
   1:L PR[91] R[100]mm/sec CNT100;
   1:  PR[91,1] = PR[90,1] + 33.874;
   1:  PR[91,2] = PR[90,2] + 9.658;
   1:L PR[91] R[100]mm/sec CNT100;
   1:  PR[91,1] = PR[90,1] + 32.240;
   1:  PR[91,2] = PR[90,2] + 11.781;
   1:L PR[91] R[100]mm/sec CNT100;
   1:  PR[91,1] = PR[90,1] + 30.188;
